KUKA KRL program: MyProgram_303().src

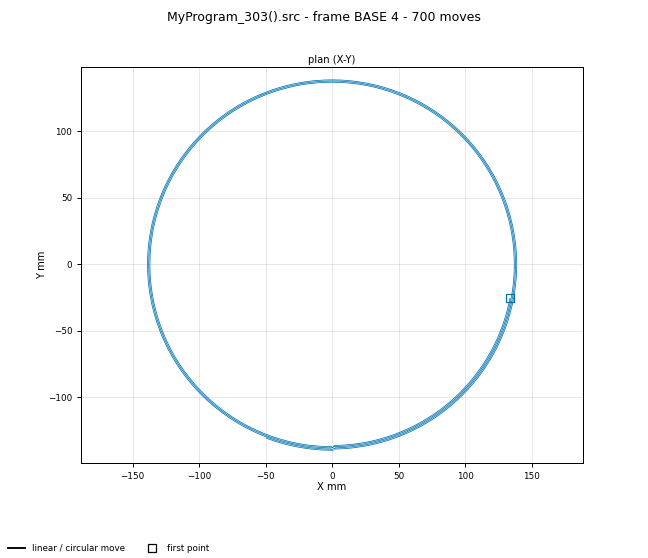
[picture p0: tool path of MyProgram_303().src in frame BASE 4, 700 of 700 moves have a stored position in this frame; points joined in program order, loops and branches not executed]
&ACCESS RVP
&REL 1
&PARAM TEMPLATE = C:\KRC\Roboter\Template\vorgabe
&PARAM EDITMASK = *
DEF MyProgram_303()
; ---- Setting reference (Base) ----
$BASE = BASE_DATA[4]

; --------------------------
; ---- Setting tool (TCP) ----
$TOOL = TOOL_DATA[3]
; --------------------------

$VEL.CP = VEL_APROX_PRINT
Startdeposition()
$VEL.CP = VEL_PRINT
LIN {X 133.6674,Y -25.5337,Z 180,A -8.434,B 5.5878,C 0.2694,E1 5.7512,E2 460.8731} C_DIS
LIN {X 132.8388,Y -29.5533,Z 180,A -10.1187,B 5.5876,C 0.2736,E1 5.7502,E2 462.5539} C_DIS
LIN {X 131.9448,Y -33.3095,Z 180,A -11.8894,B 5.5873,C 0.2804,E1 5.749,E2 464.3442} C_DIS
LIN {X 130.5853,Y -38.2938,Z 180,A -13.8432,B 5.5872,C 0.283,E1 5.7475,E2 466.272} C_DIS
LIN {X 129.5921,Y -41.5309,Z 180,A -15.2343,B 5.587,C 0.2864,E1 5.7464,E2 467.66} C_DIS
LIN {X 127.7254,Y -46.9659,Z 180,A -17.711,B 5.5866,C 0.2938,E1 5.7441,E2 470.1461} C_DIS
LIN {X 125.6978,Y -52.1446,Z 180,A -19.6502,B 5.5866,C 0.294,E1 5.7421,E2 472.0364} C_DIS
LIN {X 124,Y -56.0639,Z 180,A -21.5952,B 5.5862,C 0.3009,E1 5.7399,E2 474.0017} C_DIS
LIN {X 122.3109,Y -59.6596,Z 180,A -23.4453,B 5.5859,C 0.308,E1 5.7376,E2 475.8758} C_DIS
LIN {X 119.5176,Y -65.0767,Z 180,A -25.5702,B 5.5859,C 0.308,E1 5.735,E2 477.947} C_DIS
LIN {X 117.9855,Y -67.8162,Z 180,A -27.1675,B 5.5854,C 0.3154,E1 5.7327,E2 479.5806} C_DIS
LIN {X 115.6089,Y -71.7915,Z 180,A -28.9992,B 5.5853,C 0.3185,E1 5.7301,E2 481.3991} C_DIS
LIN {X 113.3177,Y -75.3564,Z 180,A -30.7531,B 5.585,C 0.3224,E1 5.7274,E2 483.1508} C_DIS
LIN {X 110.9133,Y -78.853,Z 180,A -32.56,B 5.5848,C 0.3269,E1 5.7245,E2 484.9618} C_DIS
LIN {X 108.1869,Y -82.5532,Z 180,A -34.4234,B 5.5846,C 0.3304,E1 5.7214,E2 486.8179} C_DIS
LIN {X 105.3409,Y -86.1552,Z 180,A -36.3118,B 5.5844,C 0.3341,E1 5.7181,E2 488.7023} C_DIS
LIN {X 102.5066,Y -89.5088,Z 180,A -38.1546,B 5.5841,C 0.3382,E1 5.7147,E2 490.546} C_DIS
LIN {X 98.895,Y -93.4837,Z 180,A -40.3296,B 5.5839,C 0.3418,E1 5.7106,E2 492.7121} C_DIS
LIN {X 95.7,Y -96.7524,Z 180,A -42.7451,B 5.5832,C 0.353,E1 5.7057,E2 495.1915} C_DIS
LIN {X 92.0984,Y -100.1859,Z 180,A -44.2158,B 5.5835,C 0.3481,E1 5.7029,E2 496.5848} C_DIS
LIN {X 89.5417,Y -102.4779,Z 180,A -45.5637,B 5.5835,C 0.3495,E1 5.7001,E2 497.9215} C_DIS
LIN {X 86.5764,Y -104.9954,Z 180,A -47.3133,B 5.5831,C 0.3543,E1 5.6963,E2 499.6868} C_DIS
LIN {X 83.034,Y -107.819,Z 180,A -49.2331,B 5.5829,C 0.358,E1 5.6921,E2 501.6099} C_DIS
LIN {X 79.3501,Y -110.5578,Z 180,A -51.1319,B 5.5827,C 0.3609,E1 5.6878,E2 503.5058} C_DIS
LIN {X 75.6563,Y -113.1174,Z 180,A -52.9009,B 5.5826,C 0.3624,E1 5.6838,E2 505.2607} C_DIS
LIN {X 72.317,Y -115.2815,Z 180,A -54.5739,B 5.5824,C 0.3651,E1 5.6798,E2 506.9348} C_DIS
LIN {X 68.7134,Y -117.4647,Z 180,A -56.3441,B 5.5822,C 0.3678,E1 5.6756,E2 508.7059} C_DIS
LIN {X 64.8663,Y -119.6324,Z 180,A -58.2317,B 5.582,C 0.3709,E1 5.6709,E2 510.5987} C_DIS
LIN {X 61.4457,Y -121.4224,Z 180,A -59.7189,B 5.582,C 0.3713,E1 5.6673,E2 512.0694} C_DIS
LIN {X 57.8895,Y -123.1589,Z 180,A -61.3233,B 5.582,C 0.3727,E1 5.6633,E2 513.6671} C_DIS
LIN {X 54.334,Y -124.7671,Z 180,A -63.1891,B 5.5816,C 0.3778,E1 5.6584,E2 515.5626} C_DIS
LIN {X 46.4604,Y -127.9079,Z 180,A -66.358,B 5.5816,C 0.3764,E1 5.6503,E2 518.6828} C_DIS
LIN {X 42.8157,Y -129.1734,Z 180,A -68.124,B 5.5814,C 0.3801,E1 5.6456,E2 520.4682} C_DIS
LIN {X 39.517,Y -130.2207,Z 180,A -69.541,B 5.5814,C 0.3809,E1 5.6418,E2 521.881} C_DIS
LIN {X 36.4352,Y -131.1162,Z 180,A -70.9127,B 5.5813,C 0.3824,E1 5.6381,E2 523.2562} C_DIS
LIN {X 32.8836,Y -132.0529,Z 180,A -72.4265,B 5.5813,C 0.3832,E1 5.634,E2 524.7669} C_DIS
LIN {X 29.4041,Y -132.8715,Z 180,A -74.0382,B 5.581,C 0.3858,E1 5.6296,E2 526.3933} C_DIS
LIN {X 25.5906,Y -133.6566,Z 180,A -75.5921,B 5.581,C 0.3858,E1 5.6254,E2 527.9372} C_DIS
LIN {X 20.5785,Y -134.5197,Z 180,A -77.875,B 5.5808,C 0.3889,E1 5.619,E2 530.2394} C_DIS
LIN {X 17.296,Y -134.9814,Z 180,A -79.1694,B 5.5808,C 0.3883,E1 5.6155,E2 531.5218} C_DIS
LIN {X 8.8845,Y -135.7952,Z 180,A -82.5567,B 5.5809,C 0.3874,E1 5.6061,E2 534.8892} C_DIS
LIN {X 1.7004,Y -136.0752,Z 180,A -85.7728,B 5.5807,C 0.3905,E1 5.5971,E2 538.1311} C_DIS
LIN {X 1.7004,Y -136.0752,Z 180,A -85.7728,B 5.5807,C 0.3905,E1 5.5971,E2 538.1311} C_DIS
Enddeposition()
LIN {X 0.9629,Y -136.9801,Z 180,A -85.7145,B 5.5127,C 0.3881,E1 5.5292,E2 538.0775} C_DIS
Startdeposition()
$VEL.CP = VEL_PRINT
LIN {X 5.9591,Y -136.8588,Z 180,A -82.9076,B 5.5134,C 0.3786,E1 5.5373,E2 535.1764} C_DIS
LIN {X 9.2064,Y -136.6797,Z 180,A -81.1696,B 5.5137,C 0.3733,E1 5.5423,E2 533.388} C_DIS
LIN {X 14.3385,Y -136.2351,Z 180,A -79.6594,B 5.5132,C 0.3808,E1 5.5462,E2 531.9612} C_DIS
LIN {X 22.708,Y -135.0919,Z 180,A -76.1483,B 5.5133,C 0.3792,E1 5.5559,E2 528.4512} C_DIS
LIN {X 26.5585,Y -134.39,Z 180,A -74.4021,B 5.5135,C 0.3767,E1 5.5608,E2 526.6898} C_DIS
LIN {X 30.3798,Y -133.5759,Z 180,A -72.9197,B 5.5135,C 0.3775,E1 5.5648,E2 525.2262} C_DIS
LIN {X 33.4089,Y -132.8509,Z 180,A -71.7147,B 5.5135,C 0.3778,E1 5.568,E2 524.033} C_DIS
LIN {X 36.6138,Y -132.0035,Z 180,A -70.25,B 5.5135,C 0.3756,E1 5.572,E2 522.5573} C_DIS
LIN {X 39.7265,Y -131.1006,Z 180,A -68.8635,B 5.5137,C 0.3739,E1 5.5757,E2 521.1658} C_DIS
LIN {X 43.1088,Y -130.0272,Z 180,A -67.3618,B 5.5137,C 0.3722,E1 5.5797,E2 519.6608} C_DIS
LIN {X 46.2144,Y -128.9561,Z 180,A -64.7574,B 5.515,C 0.3537,E1 5.587,E2 516.8931} C_DIS
LIN {X 54.4369,Y -125.706,Z 180,A -61.9666,B 5.5145,C 0.3619,E1 5.5938,E2 514.2199} C_DIS
LIN {X 58.316,Y -123.9567,Z 180,A -60.5223,B 5.5143,C 0.3642,E1 5.5974,E2 512.8183} C_DIS
LIN {X 61.5186,Y -122.3982,Z 180,A -59.0643,B 5.5144,C 0.3626,E1 5.601,E2 511.3634} C_DIS
LIN {X 65.241,Y -120.4562,Z 180,A -57.3435,B 5.5146,C 0.3606,E1 5.6053,E2 509.6458} C_DIS
LIN {X 68.9644,Y -118.3637,Z 180,A -55.5918,B 5.5147,C 0.3584,E1 5.6095,E2 507.8972} C_DIS
LIN {X 72.6617,Y -116.1305,Z 180,A -53.8371,B 5.5148,C 0.3563,E1 5.6136,E2 506.1478} C_DIS
LIN {X 76.146,Y -113.8758,Z 180,A -52.1006,B 5.515,C 0.3534,E1 5.6177,E2 504.4098} C_DIS
LIN {X 79.7915,Y -111.3519,Z 180,A -50.2937,B 5.5152,C 0.3508,E1 5.6218,E2 502.6076} C_DIS
LIN {X 83.4506,Y -108.637,Z 180,A -48.4066,B 5.5154,C 0.3477,E1 5.626,E2 500.7213} C_DIS
LIN {X 86.9716,Y -105.8394,Z 180,A -46.5374,B 5.5156,C 0.3443,E1 5.6301,E2 498.8521} C_DIS
LIN {X 91.926,Y -101.5655,Z 180,A -43.4145,B 5.5163,C 0.3333,E1 5.6367,E2 495.6763} C_DIS
LIN {X 95.3245,Y -98.3827,Z 180,A -41.896,B 5.5161,C 0.3356,E1 5.6397,E2 494.2123} C_DIS
LIN {X 98.0792,Y -95.6375,Z 180,A -40.532,B 5.5161,C 0.3361,E1 5.6423,E2 492.8809} C_DIS
LIN {X 102.4384,Y -90.9526,Z 180,A -37.732,B 5.5166,C 0.3285,E1 5.6476,E2 490.0626} C_DIS
LIN {X 105.2335,Y -87.7041,Z 180,A -35.9364,B 5.5168,C 0.3244,E1 5.6509,E2 488.2651} C_DIS
LIN {X 108.1029,Y -84.1413,Z 180,A -34.0819,B 5.517,C 0.3209,E1 5.6541,E2 486.4165} C_DIS
LIN {X 110.6826,Y -80.7183,Z 180,A -32.3179,B 5.5172,C 0.3171,E1 5.657,E2 484.6547} C_DIS
LIN {X 113.2996,Y -77.0011,Z 180,A -30.4716,B 5.5174,C 0.3134,E1 5.6599,E2 482.8138} C_DIS
LIN {X 115.7618,Y -73.2472,Z 180,A -28.6372,B 5.5177,C 0.3095,E1 5.6627,E2 480.9833} C_DIS
LIN {X 118.1004,Y -69.4134,Z 180,A -26.8055,B 5.5179,C 0.3055,E1 5.6653,E2 479.1559} C_DIS
LIN {X 120.3903,Y -65.3619,Z 180,A -24.5644,B 5.5184,C 0.2961,E1 5.6684,E2 476.8748} C_DIS
LIN {X 122.2336,Y -61.8418,Z 180,A -23.335,B 5.5183,C 0.2984,E1 5.6699,E2 475.7} C_DIS
LIN {X 124.2076,Y -57.7748,Z 180,A -21.3722,B 5.5186,C 0.2923,E1 5.6722,E2 473.7262} C_DIS
LIN {X 126.0977,Y -53.5294,Z 180,A -19.5105,B 5.5188,C 0.2885,E1 5.6743,E2 471.8735} C_DIS
LIN {X 127.5825,Y -49.8816,Z 180,A -18.0664,B 5.5188,C 0.2872,E1 5.6757,E2 470.4541} C_DIS
LIN {X 128.8042,Y -46.636,Z 180,A -16.4286,B 5.5192,C 0.2804,E1 5.6773,E2 468.7908} C_DIS
LIN {X 130.343,Y -42.1468,Z 180,A -14.6249,B 5.5193,C 0.2777,E1 5.6789,E2 467.0087} C_DIS
LIN {X 131.2957,Y -39.0797,Z 180,A -13.4462,B 5.5193,C 0.2766,E1 5.6799,E2 465.8501} C_DIS
LIN {X 132.2472,Y -35.7252,Z 180,A -12.0475,B 5.5196,C 0.2735,E1 5.6809,E2 464.4578} C_DIS
LIN {X 133.1587,Y -32.1591,Z 180,A -10.4265,B 5.5198,C 0.2679,E1 5.682,E2 462.825} C_DIS
LIN {X 133.9191,Y -28.829,Z 180,A -9.0632,B 5.52,C 0.2649,E1 5.6828,E2 461.4688} C_DIS
LIN {X 135.0379,Y -23.032,Z 180,A -6.3047,B 5.5205,C 0.2535,E1 5.6842,E2 458.6711} C_DIS
LIN {X 135.5799,Y -19.5857,Z 180,A -5.0968,B 5.5205,C 0.2533,E1 5.6847,E2 457.4944} C_DIS
LIN {X 136.2099,Y -14.5726,Z 180,A -2.5529,B 5.5211,C 0.2406,E1 5.6855,E2 454.8933} C_DIS
LIN {X 136.6579,Y -9.505,Z 180,A -1.0891,B 5.5209,C 0.2448,E1 5.6858,E2 453.5132} C_DIS
LIN {X 136.8714,Y -5.6402,Z 180,A 0.5488,B 5.5211,C 0.2399,E1 5.686,E2 451.8716} C_DIS
LIN {X 136.9726,Y -2.0268,Z 180,A 2.7438,B 5.5217,C 0.225,E1 5.6861,E2 449.5877} C_DIS
LIN {X 136.9301,Y 3.962,Z 180,A 4.4252,B 5.5215,C 0.2307,E1 5.6861,E2 448.0102} C_DIS
LIN {X 136.5326,Y 11.157,Z 180,A 7.2664,B 5.5217,C 0.2248,E1 5.6855,E2 445.1889} C_DIS
LIN {X 135.9491,Y 16.8438,Z 180,A 9.7561,B 5.5221,C 0.2165,E1 5.6848,E2 442.685} C_DIS
LIN {X 135.4199,Y 20.6637,Z 180,A 11.3418,B 5.5222,C 0.2123,E1 5.6841,E2 441.1017} C_DIS
LIN {X 134.6933,Y 24.9749,Z 180,A 13.1664,B 5.5224,C 0.2073,E1 5.6832,E2 439.2764} C_DIS
LIN {X 133.926,Y 28.7974,Z 180,A 14.6505,B 5.5225,C 0.205,E1 5.6824,E2 437.8097} C_DIS
LIN {X 133.2251,Y 31.8835,Z 180,A 15.9603,B 5.5226,C 0.2015,E1 5.6816,E2 436.5008} C_DIS
LIN {X 132.3877,Y 35.1986,Z 180,A 17.271,B 5.5227,C 0.1994,E1 5.6807,E2 435.2044} C_DIS
LIN {X 131.4832,Y 38.4392,Z 180,A 18.6758,B 5.5229,C 0.1956,E1 5.6796,E2 433.799} C_DIS
LIN {X 130.378,Y 42.0372,Z 180,A 20.3219,B 5.523,C 0.1902,E1 5.6782,E2 432.1429} C_DIS
LIN {X 129.086,Y 45.8542,Z 180,A 21.9681,B 5.5232,C 0.1863,E1 5.6767,E2 430.5007} C_DIS
LIN {X 127.6955,Y 49.5908,Z 180,A 23.4129,B 5.5232,C 0.1852,E1 5.6753,E2 429.0831} C_DIS
LIN {X 126.4948,Y 52.5784,Z 180,A 24.9531,B 5.5234,C 0.1787,E1 5.6736,E2 427.5177} C_DIS
LIN {X 124.5309,Y 57.0756,Z 180,A 26.8317,B 5.5235,C 0.176,E1 5.6715,E2 425.6601} C_DIS
LIN {X 123.0141,Y 60.2746,Z 180,A 28.2274,B 5.5235,C 0.1735,E1 5.6698,E2 424.2744} C_DIS
LIN {X 121.4029,Y 63.4566,Z 180,A 29.7193,B 5.5237,C 0.1697,E1 5.6679,E2 422.7817} C_DIS
LIN {X 119.27,Y 67.3845,Z 180,A 31.6372,B 5.5239,C 0.1643,E1 5.6653,E2 420.857} C_DIS
LIN {X 117.0777,Y 71.1253,Z 180,A 33.4111,B 5.5239,C 0.1605,E1 5.6628,E2 419.0873} C_DIS
LIN {X 114.7348,Y 74.846,Z 180,A 35.1874,B 5.5241,C 0.157,E1 5.6601,E2 417.3181} C_DIS
LIN {X 112.2574,Y 78.513,Z 180,A 37.0342,B 5.5241,C 0.1527,E1 5.6572,E2 415.4712} C_DIS
LIN {X 109.5754,Y 82.2149,Z 180,A 38.7169,B 5.5242,C 0.1517,E1 5.6544,E2 413.8165} C_DIS
LIN {X 107.2012,Y 85.2866,Z 180,A 40.3892,B 5.5243,C 0.1473,E1 5.6516,E2 412.1376} C_DIS
LIN {X 104.7567,Y 88.2725,Z 180,A 42.0713,B 5.5245,C 0.1428,E1 5.6485,E2 410.4466} C_DIS
LIN {X 101.7751,Y 91.6946,Z 180,A 43.8321,B 5.5245,C 0.1407,E1 5.6453,E2 408.7024} C_DIS
LIN {X 98.7669,Y 94.9271,Z 180,A 45.7626,B 5.5246,C 0.1356,E1 5.6416,E2 406.7611} C_DIS
LIN {X 95.5482,Y 98.1661,Z 180,A 47.3451,B 5.5246,C 0.1364,E1 5.6385,E2 405.2189} C_DIS
LIN {X 92.6799,Y 100.8779,Z 180,A 49.211,B 5.5248,C 0.1302,E1 5.6347,E2 403.3259} C_DIS
LIN {X 89.3728,Y 103.8191,Z 180,A 51.0246,B 5.5248,C 0.1272,E1 5.6309,E2 401.5167} C_DIS
LIN {X 85.8701,Y 106.7346,Z 180,A 52.941,B 5.5249,C 0.1236,E1 5.6267,E2 399.5988} C_DIS
LIN {X 82.2251,Y 109.5677,Z 180,A 54.8506,B 5.5249,C 0.1205,E1 5.6225,E2 397.6917} C_DIS
LIN {X 78.6371,Y 112.1708,Z 180,A 56.653,B 5.525,C 0.1181,E1 5.6184,E2 395.8955} C_DIS
LIN {X 75.107,Y 114.5641,Z 180,A 58.4111,B 5.525,C 0.1156,E1 5.6143,E2 394.1405} C_DIS
LIN {X 71.3198,Y 116.9596,Z 180,A 60.281,B 5.5252,C 0.1128,E1 5.6099,E2 392.2711} C_DIS
LIN {X 67.5354,Y 119.1849,Z 180,A 62.1056,B 5.5252,C 0.1103,E1 5.6055,E2 390.448} C_DIS
LIN {X 63.8288,Y 121.2075,Z 180,A 63.7161,B 5.5252,C 0.11,E1 5.6016,E2 388.8567} C_DIS
LIN {X 61.2437,Y 122.536,Z 180,A 65.023,B 5.5252,C 0.1072,E1 5.5983,E2 387.5387} C_DIS
LIN {X 57.8222,Y 124.1857,Z 180,A 66.5177,B 5.5252,C 0.1064,E1 5.5945,E2 386.0557} C_DIS
LIN {X 54.6205,Y 125.6266,Z 180,A 67.9197,B 5.5252,C 0.1056,E1 5.591,E2 384.662} C_DIS
LIN {X 51.4939,Y 126.9403,Z 180,A 69.2666,B 5.5253,C 0.1049,E1 5.5875,E2 383.3242} C_DIS
LIN {X 48.8881,Y 127.9683,Z 180,A 70.6345,B 5.5253,C 0.1011,E1 5.5839,E2 381.9322} C_DIS
LIN {X 45.08,Y 129.357,Z 180,A 72.0835,B 5.5253,C 0.1027,E1 5.5801,E2 380.5139} C_DIS
LIN {X 42.0821,Y 130.3636,Z 180,A 73.4942,B 5.5253,C 0.1003,E1 5.5764,E2 379.0926} C_DIS
LIN {X 37.472,Y 131.7635,Z 180,A 75.439,B 5.5254,C 0.0995,E1 5.5712,E2 377.1569} C_DIS
LIN {X 33.9468,Y 132.7144,Z 180,A 77.0132,B 5.5254,C 0.0978,E1 5.5669,E2 375.5773} C_DIS
LIN {X 30.7155,Y 133.4992,Z 180,A 78.447,B 5.5254,C 0.0962,E1 5.563,E2 374.1385} C_DIS
LIN {X 27.37,Y 134.2249,Z 180,A 79.87,B 5.5254,C 0.0955,E1 5.5591,E2 372.7169} C_DIS
LIN {X 23.2032,Y 135.0093,Z 180,A 81.6985,B 5.5255,C 0.0938,E1 5.5541,E2 370.8823} C_DIS
LIN {X 19.1357,Y 135.6442,Z 180,A 83.6361,B 5.5255,C 0.0904,E1 5.5487,E2 368.9186} C_DIS
LIN {X 15.5832,Y 136.0995,Z 180,A 85.2933,B 5.5256,C 0.0879,E1 5.544,E2 367.2422} C_DIS
LIN {X 11.3245,Y 136.5185,Z 180,A 86.6921,B 5.5256,C 0.0922,E1 5.5402,E2 365.8924} C_DIS
LIN {X 8.4551,Y 136.7261,Z 180,A 88.5823,B 5.5256,C 0.0836,E1 5.5348,E2 363.9176} C_DIS
LIN {X 2.4594,Y 136.9654,Z 180,A 90.6298,B 5.5256,C 0.0889,E1 5.5292,E2 361.9286} C_DIS
LIN {X -1.0774,Y 136.9835,Z 180,A 91.8821,B 5.5256,C 0.0916,E1 5.5258,E2 360.7051} C_DIS
LIN {X -5.2438,Y 136.8869,Z 180,A 93.5421,B 5.5256,C 0.0927,E1 5.5212,E2 359.056} C_DIS
LIN {X -10.5015,Y 136.5851,Z 180,A 95.9583,B 5.5256,C 0.0905,E1 5.5144,E2 356.6147} C_DIS
LIN {X -16.7957,Y 135.9548,Z 180,A 98.4644,B 5.5256,C 0.0928,E1 5.5074,E2 354.1271} C_DIS
LIN {X -20.631,Y 135.425,Z 180,A 100.0493,B 5.5256,C 0.0938,E1 5.5031,E2 352.5474} C_DIS
LIN {X -24.1026,Y 134.85,Z 180,A 101.5008,B 5.5255,C 0.0947,E1 5.4991,E2 351.0991} C_DIS
LIN {X -27.7276,Y 134.1522,Z 180,A 103.0718,B 5.5255,C 0.0952,E1 5.4948,E2 349.5258} C_DIS
LIN {X -31.8835,Y 133.2251,Z 180,A 104.7738,B 5.5255,C 0.0972,E1 5.4902,E2 347.8345} C_DIS
LIN {X -34.9603,Y 132.4512,Z 180,A 105.9658,B 5.5255,C 0.0996,E1 5.487,E2 346.6599} C_DIS
LIN {X -37.8601,Y 131.6528,Z 180,A 107.5127,B 5.5255,C 0.0973,E1 5.4827,E2 345.0784} C_DIS
LIN {X -41.5721,Y 130.5265,Z 180,A 109.0374,B 5.5255,C 0.0997,E1 5.4787,E2 343.5667} C_DIS
LIN {X -48.3571,Y 128.1682,Z 180,A 112.1227,B 5.5254,C 0.1016,E1 5.4706,E2 340.4736} C_DIS
LIN {X -51.0775,Y 127.1082,Z 180,A 113.5748,B 5.5254,C 0.1004,E1 5.4667,E2 338.9938} C_DIS
LIN {X -55.22,Y 125.3664,Z 180,A 115.3255,B 5.5254,C 0.1038,E1 5.4623,E2 337.2605} C_DIS
LIN {X -58.7178,Y 123.7648,Z 180,A 116.8367,B 5.5253,C 0.1068,E1 5.4585,E2 335.7624} C_DIS
LIN {X -61.8768,Y 122.2159,Z 180,A 118.3402,B 5.5253,C 0.1083,E1 5.4547,E2 334.2561} C_DIS
LIN {X -65.0139,Y 120.5784,Z 180,A 119.9047,B 5.5253,C 0.1093,E1 5.4509,E2 332.6824} C_DIS
LIN {X -68.9535,Y 118.3701,Z 180,A 121.8521,B 5.5252,C 0.1113,E1 5.4461,E2 330.7292} C_DIS
LIN {X -71.6444,Y 116.7604,Z 180,A 123.3661,B 5.5252,C 0.1112,E1 5.4425,E2 329.1912} C_DIS
LIN {X -74.4018,Y 115.0232,Z 180,A 124.5687,B 5.5252,C 0.1149,E1 5.4397,E2 328.0095} C_DIS
LIN {X -77.9872,Y 112.6233,Z 180,A 126.4212,B 5.5251,C 0.1173,E1 5.4354,E2 326.1525} C_DIS
LIN {X -81.7444,Y 109.9262,Z 180,A 128.3434,B 5.525,C 0.1206,E1 5.4311,E2 324.2334} C_DIS
LIN {X -85.3449,Y 107.1549,Z 180,A 130.2501,B 5.525,C 0.1238,E1 5.4269,E2 322.3274} C_DIS
LIN {X -88.6469,Y 104.4397,Z 180,A 132.1044,B 5.5249,C 0.1264,E1 5.4229,E2 320.4664} C_DIS
LIN {X -92.1385,Y 101.3727,Z 180,A 134.0526,B 5.5248,C 0.13,E1 5.4188,E2 318.5193} C_DIS
LIN {X -95.4202,Y 98.29,Z 180,A 135.9744,B 5.5247,C 0.1334,E1 5.4149,E2 316.5944} C_DIS
LIN {X -98.6326,Y 95.0664,Z 180,A 137.9163,B 5.5247,C 0.1368,E1 5.4111,E2 314.6493} C_DIS
LIN {X -101.6556,Y 91.8267,Z 180,A 139.8184,B 5.5245,C 0.1402,E1 5.4075,E2 312.7428} C_DIS
LIN {X -104.4792,Y 88.6004,Z 180,A 141.6551,B 5.5245,C 0.1437,E1 5.4042,E2 310.9022} C_DIS
LIN {X -107.4064,Y 85.0288,Z 180,A 143.6482,B 5.5243,C 0.1474,E1 5.4007,E2 308.9031} C_DIS
LIN {X -110.091,Y 81.5231,Z 180,A 145.5103,B 5.5243,C 0.1514,E1 5.3976,E2 307.0408} C_DIS
LIN {X -112.678,Y 77.9086,Z 180,A 147.4126,B 5.5241,C 0.1553,E1 5.3945,E2 305.1348} C_DIS
LIN {X -114.279,Y 75.54,Z 180,A 148.6489,B 5.5241,C 0.1578,E1 5.3926,E2 303.8945} C_DIS
LIN {X -117.1143,Y 71.0648,Z 180,A 150.8875,B 5.5239,C 0.1629,E1 5.3893,E2 301.655} C_DIS
LIN {X -119.3249,Y 67.2869,Z 180,A 152.7732,B 5.5238,C 0.167,E1 5.3866,E2 299.7641} C_DIS
LIN {X -121.5025,Y 63.267,Z 180,A 155.0178,B 5.5238,C 0.1687,E1 5.3837,E2 297.4796} C_DIS
LIN {X -123.2185,Y 59.8602,Z 180,A 156.3404,B 5.5235,C 0.1753,E1 5.3821,E2 296.1927} C_DIS
LIN {X -124.8727,Y 56.3238,Z 180,A 157.9398,B 5.5234,C 0.1798,E1 5.3802,E2 294.5988} C_DIS
LIN {X -126.2063,Y 53.2692,Z 180,A 159.4289,B 5.5233,C 0.1826,E1 5.3786,E2 293.0991} C_DIS
LIN {X -127.6676,Y 49.6625,Z 180,A 161.0329,B 5.5231,C 0.1872,E1 5.3769,E2 291.4994} C_DIS
LIN {X -130.2229,Y 42.521,Z 180,A 164.4398,B 5.5229,C 0.1936,E1 5.3738,E2 288.0662} C_DIS
LIN {X -132.1707,Y 36.0121,Z 180,A 167.3523,B 5.5227,C 0.2008,E1 5.3715,E2 285.1473} C_DIS
LIN {X -133.1847,Y 32.0508,Z 180,A 168.8875,B 5.5224,C 0.2071,E1 5.3705,E2 283.6354} C_DIS
LIN {X -133.8797,Y 29.0117,Z 180,A 170.3023,B 5.5224,C 0.2097,E1 5.3696,E2 282.2078} C_DIS
LIN {X -134.5787,Y 25.5743,Z 180,A 171.826,B 5.5222,C 0.2133,E1 5.3688,E2 280.6782} C_DIS
LIN {X -135.3067,Y 21.3955,Z 180,A 173.6561,B 5.522,C 0.2178,E1 5.368,E2 278.8427} C_DIS
LIN {X -135.7841,Y 18.1179,Z 180,A 175.094,B 5.5219,C 0.2212,E1 5.3674,E2 277.3993} C_DIS
LIN {X -136.2011,Y 14.6539,Z 180,A 176.5536,B 5.5217,C 0.2254,E1 5.3669,E2 275.9408} C_DIS
LIN {X -136.5505,Y 10.9457,Z 180,A 178.2214,B 5.5216,C 0.2288,E1 5.3665,E2 274.2605} C_DIS
LIN {X -136.8207,Y 6.7542,Z 180,A 179.9883,B 5.5214,C 0.2337,E1 5.3663,E2 272.4936} C_DIS
LIN {X -136.9645,Y 2.5098,Z 180,A -178.198,B 5.5212,C 0.2385,E1 5.3661,E2 270.6767} C_DIS
LIN {X -136.9795,Y -1.6063,Z 180,A -176.3484,B 5.521,C 0.2422,E1 5.3661,E2 268.8123} C_DIS
LIN {X -136.8732,Y -5.5952,Z 180,A -174.6513,B 5.5208,C 0.2467,E1 5.3663,E2 267.1127} C_DIS
LIN {X -136.6367,Y -9.7954,Z 180,A -172.9278,B 5.5206,C 0.252,E1 5.3666,E2 265.3951} C_DIS
LIN {X -136.3486,Y -13.2123,Z 180,A -171.4508,B 5.5204,C 0.2557,E1 5.367,E2 263.9137} C_DIS
LIN {X -135.9321,Y -16.9858,Z 180,A -169.7822,B 5.5202,C 0.2595,E1 5.3675,E2 262.2361} C_DIS
LIN {X -135.4106,Y -20.7242,Z 180,A -168.1633,B 5.52,C 0.2635,E1 5.3682,E2 260.6132} C_DIS
LIN {X -134.8324,Y -24.201,Z 180,A -166.6195,B 5.5199,C 0.267,E1 5.3689,E2 259.0616} C_DIS
LIN {X -133.9847,Y -28.5252,Z 180,A -164.7599,B 5.5196,C 0.272,E1 5.37,E2 257.2011} C_DIS
LIN {X -133.2114,Y -31.9403,Z 180,A -163.083,B 5.5196,C 0.2741,E1 5.3711,E2 255.4982} C_DIS
LIN {X -131.3234,Y -38.985,Z 180,A -160.0565,B 5.5191,C 0.2826,E1 5.3733,E2 252.4767} C_DIS
LIN {X -130.053,Y -43.0312,Z 180,A -158.5073,B 5.5187,C 0.2895,E1 5.3746,E2 250.9571} C_DIS
LIN {X -128.3114,Y -47.9748,Z 180,A -156.0573,B 5.5186,C 0.2929,E1 5.377,E2 248.4756} C_DIS
LIN {X -127.1245,Y -51.0369,Z 180,A -154.6333,B 5.5184,C 0.296,E1 5.3784,E2 247.0459} C_DIS
LIN {X -125.7124,Y -54.4222,Z 180,A -153.1744,B 5.5181,C 0.3007,E1 5.38,E2 245.5974} C_DIS
LIN {X -124.3954,Y -57.3686,Z 180,A -151.6856,B 5.5181,C 0.3029,E1 5.3818,E2 244.0916} C_DIS
LIN {X -122.5724,Y -61.17,Z 180,A -149.85,B 5.5178,C 0.3066,E1 5.384,E2 242.2477} C_DIS
LIN {X -120.6186,Y -64.939,Z 180,A -148.0859,B 5.5176,C 0.3111,E1 5.3863,E2 240.4858} C_DIS
LIN {X -118.3791,Y -68.9379,Z 180,A -146.0638,B 5.5174,C 0.3148,E1 5.3891,E2 238.4512} C_DIS
LIN {X -116.1088,Y -72.6967,Z 180,A -144.1651,B 5.5171,C 0.3186,E1 5.3919,E2 236.5453} C_DIS
LIN {X -113.6973,Y -76.4135,Z 180,A -142.2344,B 5.5169,C 0.3221,E1 5.3949,E2 234.6054} C_DIS
LIN {X -111.1285,Y -80.1031,Z 180,A -140.3205,B 5.5167,C 0.326,E1 5.398,E2 232.6878} C_DIS
LIN {X -108.3692,Y -83.7977,Z 180,A -138.3801,B 5.5165,C 0.3302,E1 5.4013,E2 230.7466} C_DIS
LIN {X -105.4348,Y -87.461,Z 180,A -136.3998,B 5.5162,C 0.3342,E1 5.4048,E2 228.7647} C_DIS
LIN {X -102.7591,Y -90.5898,Z 180,A -134.1066,B 5.5163,C 0.332,E1 5.4092,E2 226.3979} C_DIS
LIN {X -99.379,Y -94.2859,Z 180,A -132.4987,B 5.5158,C 0.3412,E1 5.4121,E2 224.8538} C_DIS
LIN {X -96.1662,Y -97.5607,Z 180,A -130.5157,B 5.5156,C 0.3443,E1 5.416,E2 222.8629} C_DIS
LIN {X -93.0223,Y -100.5632,Z 180,A -128.6509,B 5.5154,C 0.3472,E1 5.4198,E2 220.9924} C_DIS
LIN {X -90.2215,Y -103.0826,Z 180,A -126.9158,B 5.5154,C 0.3484,E1 5.4235,E2 219.237} C_DIS
LIN {X -86.1573,Y -106.5029,Z 180,A -124.839,B 5.515,C 0.3537,E1 5.428,E2 217.1793} C_DIS
LIN {X -82.6996,Y -109.2096,Z 180,A -122.9697,B 5.5148,C 0.3564,E1 5.4321,E2 215.3059} C_DIS
LIN {X -79.1565,Y -111.8044,Z 180,A -121.121,B 5.5147,C 0.3592,E1 5.4363,E2 213.4558} C_DIS
LIN {X -75.775,Y -114.1235,Z 180,A -119.3511,B 5.5145,C 0.3612,E1 5.4404,E2 211.6788} C_DIS
LIN {X -72.1149,Y -116.4708,Z 180,A -117.5251,B 5.5144,C 0.3637,E1 5.4447,E2 209.852} C_DIS
LIN {X -68.2672,Y -118.7674,Z 180,A -115.5976,B 5.5142,C 0.3656,E1 5.4494,E2 207.9175} C_DIS
LIN {X -64.39,Y -120.9129,Z 180,A -113.7925,B 5.514,C 0.3685,E1 5.4538,E2 206.1186} C_DIS
LIN {X -61.2254,Y -122.5451,Z 180,A -112.2197,B 5.514,C 0.3693,E1 5.4578,E2 204.5348} C_DIS
LIN {X -57.8098,Y -124.1914,Z 180,A -110.7347,B 5.5138,C 0.3722,E1 5.4615,E2 203.0628} C_DIS
LIN {X -54.9048,Y -125.5037,Z 180,A -109.3801,B 5.5138,C 0.3733,E1 5.4649,E2 201.7053} C_DIS
LIN {X -52.0165,Y -126.7289,Z 180,A -107.9405,B 5.5138,C 0.3732,E1 5.4687,E2 200.249} C_DIS
LIN {X -48.2267,Y -128.217,Z 180,A -106.4581,B 5.5135,C 0.3772,E1 5.4725,E2 198.7949} C_DIS
LIN {X -45.7391,Y -129.1275,Z 180,A -105.0653,B 5.5136,C 0.3749,E1 5.4763,E2 197.3648} C_DIS
LIN {X -40.6777,Y -130.8094,Z 180,A -103.0524,B 5.5133,C 0.3791,E1 5.4815,E2 195.3799} C_DIS
LIN {X -37.0885,Y -131.8708,Z 180,A -101.3685,B 5.5133,C 0.3788,E1 5.4861,E2 193.6802} C_DIS
LIN {X -33.9468,Y -132.7144,Z 180,A -99.9951,B 5.5133,C 0.3795,E1 5.4898,E2 192.3047} C_DIS
LIN {X -30.5974,Y -133.5262,Z 180,A -98.5685,B 5.5133,C 0.3804,E1 5.4937,E2 190.8797} C_DIS
LIN {X -26.8584,Y -134.329,Z 180,A -96.8584,B 5.5133,C 0.3798,E1 5.4984,E2 189.1547} C_DIS
LIN {X -23.1372,Y -135.0203,Z 180,A -94.9328,B 5.5135,C 0.3762,E1 5.5038,E2 187.1838} C_DIS
LIN {X -19.0269,Y -135.6598,Z 180,A -93.5267,B 5.5132,C 0.3808,E1 5.5076,E2 185.8207} C_DIS
LIN {X -14.7911,Y -136.1864,Z 180,A -91.8602,B 5.5131,C 0.3826,E1 5.5122,E2 184.1691} C_DIS
LIN {X -8.7636,Y -136.7071,Z 180,A -89.1656,B 5.5132,C 0.3808,E1 5.5198,E2 181.4521} C_DIS
LIN {X -3.9799,Y -136.9296,Z 180,A -87.3425,B 5.5131,C 0.3831,E1 5.5248,E2 179.6516} C_DIS
LIN {X -0.5118,Y -136.9866,Z 180,A -85.7833,B 5.5131,C 0.3815,E1 5.5292,E2 178.0775} C_DIS
LIN {X -0.5118,Y -136.9866,Z 180,A -85.7833,B 5.5131,C 0.3815,E1 5.5292,E2 178.0775} C_DIS
Enddeposition()
LIN {X 0.9731,Y -137.885,Z 180,A -85.2998,B 5.4467,C 0.3854,E1 5.4643,E2 177.6628} C_DIS
Startdeposition()
$VEL.CP = VEL_PRINT
LIN {X -2.4494,Y -137.8683,Z 180,A -87.2819,B 5.4462,C 0.3925,E1 5.4585,E2 179.7189} C_DIS
LIN {X -6.1473,Y -137.755,Z 180,A -88.7568,B 5.4462,C 0.3918,E1 5.4544,E2 181.1864} C_DIS
LIN {X -9.2578,Y -137.581,Z 180,A -90.0542,B 5.4462,C 0.3918,E1 5.4508,E2 182.4847} C_DIS
LIN {X -13.3319,Y -137.2439,Z 180,A -91.7985,B 5.4462,C 0.3921,E1 5.4459,E2 184.2356} C_DIS
LIN {X -17.1247,Y -136.8246,Z 180,A -93.3499,B 5.4462,C 0.3914,E1 5.4416,E2 185.7833} C_DIS
LIN {X -20.3016,Y -136.3894,Z 180,A -94.688,B 5.4462,C 0.3911,E1 5.4379,E2 187.1225} C_DIS
LIN {X -23.4919,Y -135.8763,Z 180,A -96.0371,B 5.4462,C 0.3907,E1 5.4342,E2 188.473} C_DIS
LIN {X -26.1819,Y -135.3816,Z 180,A -97.2269,B 5.4462,C 0.3909,E1 5.4309,E2 189.67} C_DIS
LIN {X -29.9023,Y -134.6109,Z 180,A -98.768,B 5.4464,C 0.3897,E1 5.4267,E2 191.2068} C_DIS
LIN {X -33.1168,Y -133.8563,Z 180,A -100.1492,B 5.4464,C 0.389,E1 5.4229,E2 192.5894} C_DIS
LIN {X -36.093,Y -133.0833,Z 180,A -101.4205,B 5.4464,C 0.3882,E1 5.4195,E2 193.8603} C_DIS
LIN {X -39.55,Y -132.0986,Z 180,A -102.9413,B 5.4465,C 0.3875,E1 5.4154,E2 195.385} C_DIS
LIN {X -42.7627,Y -131.0938,Z 180,A -104.3516,B 5.4465,C 0.3866,E1 5.4117,E2 196.7971} C_DIS
LIN {X -45.9685,Y -130.0044,Z 180,A -105.7711,B 5.4466,C 0.3856,E1 5.4079,E2 198.2185} C_DIS
LIN {X -48.7145,Y -128.9982,Z 180,A -106.9979,B 5.4467,C 0.3846,E1 5.4047,E2 199.4469} C_DIS
LIN {X -52.3467,Y -127.5698,Z 180,A -108.6359,B 5.4468,C 0.3833,E1 5.4004,E2 201.0873} C_DIS
LIN {X -55.5127,Y -126.2243,Z 180,A -110.0807,B 5.4468,C 0.382,E1 5.3967,E2 202.5343} C_DIS
LIN {X -58.1961,Y -125.0073,Z 180,A -111.3622,B 5.4469,C 0.3813,E1 5.3935,E2 203.8233} C_DIS
LIN {X -61.7815,Y -123.2773,Z 180,A -112.9924,B 5.4471,C 0.3791,E1 5.3894,E2 205.4506} C_DIS
LIN {X -64.4484,Y -121.9017,Z 180,A -114.2005,B 5.4472,C 0.3772,E1 5.3864,E2 206.6537} C_DIS
LIN {X -67.9438,Y -119.9912,Z 180,A -116.0129,B 5.4472,C 0.3768,E1 5.3819,E2 208.4865} C_DIS
LIN {X -71.7292,Y -117.7674,Z 180,A -117.8623,B 5.4474,C 0.3746,E1 5.3775,E2 210.3392} C_DIS
LIN {X -75.4559,Y -115.4151,Z 180,A -119.7284,B 5.4476,C 0.3723,E1 5.3731,E2 212.2098} C_DIS
LIN {X -79.1176,Y -112.9365,Z 180,A -121.6174,B 5.4477,C 0.37,E1 5.3687,E2 214.1053} C_DIS
LIN {X -82.7078,Y -110.3343,Z 180,A -123.4818,B 5.4479,C 0.3673,E1 5.3645,E2 215.9725} C_DIS
LIN {X -86.2205,Y -107.6117,Z 180,A -125.3659,B 5.4481,C 0.3646,E1 5.3604,E2 217.8611} C_DIS
LIN {X -89.6495,Y -104.7721,Z 180,A -127.2146,B 5.4483,C 0.3614,E1 5.3564,E2 219.7094} C_DIS
LIN {X -92.9893,Y -101.8196,Z 180,A -129.1321,B 5.4485,C 0.3586,E1 5.3524,E2 221.6349} C_DIS
LIN {X -96.2342,Y -98.7583,Z 180,A -131.0195,B 5.4487,C 0.3555,E1 5.3486,E2 223.5263} C_DIS
LIN {X -99.3464,Y -95.6268,Z 180,A -132.8606,B 5.4489,C 0.3519,E1 5.345,E2 225.3678} C_DIS
LIN {X -102.4189,Y -92.3288,Z 180,A -134.7967,B 5.4491,C 0.3488,E1 5.3414,E2 227.3116} C_DIS
LIN {X -105.3492,Y -88.9707,Z 180,A -136.6529,B 5.4494,C 0.3449,E1 5.338,E2 229.1678} C_DIS
LIN {X -108.1657,Y -85.5244,Z 180,A -138.5723,B 5.4496,C 0.3416,E1 5.3346,E2 231.0956} C_DIS
LIN {X -110.8645,Y -81.9958,Z 180,A -140.4238,B 5.4498,C 0.3376,E1 5.3315,E2 232.9472} C_DIS
LIN {X -113.4422,Y -78.3907,Z 180,A -142.3043,B 5.4501,C 0.3338,E1 5.3285,E2 234.832} C_DIS
LIN {X -115.8957,Y -74.7156,Z 180,A -144.1631,B 5.4503,C 0.3297,E1 5.3256,E2 236.693} C_DIS
LIN {X -118.2225,Y -70.9766,Z 180,A -146.0824,B 5.4505,C 0.3262,E1 5.3228,E2 238.623} C_DIS
LIN {X -120.4203,Y -67.1803,Z 180,A -147.9459,B 5.4508,C 0.3221,E1 5.3202,E2 240.4908} C_DIS
LIN {X -122.4874,Y -63.3331,Z 180,A -149.6874,B 5.4511,C 0.3169,E1 5.318,E2 242.2221} C_DIS
LIN {X -123.9502,Y -60.4173,Z 180,A -151.0834,B 5.4512,C 0.3139,E1 5.3162,E2 243.6226} C_DIS
LIN {X -125.5195,Y -57.0884,Z 180,A -152.6394,B 5.4514,C 0.3103,E1 5.3144,E2 245.1813} C_DIS
LIN {X -126.9012,Y -53.9472,Z 180,A -154.0993,B 5.4516,C 0.3069,E1 5.3128,E2 246.6448} C_DIS
LIN {X -128.2105,Y -50.7574,Z 180,A -155.566,B 5.4518,C 0.3035,E1 5.3113,E2 248.1151} C_DIS
LIN {X -129.4277,Y -47.5678,Z 180,A -157.019,B 5.452,C 0.3,E1 5.3098,E2 249.5716} C_DIS
LIN {X -130.5597,Y -44.3666,Z 180,A -158.4642,B 5.4522,C 0.2966,E1 5.3085,E2 251.0204} C_DIS
LIN {X -131.5271,Y -41.4064,Z 180,A -159.803,B 5.4524,C 0.2935,E1 5.3074,E2 252.364} C_DIS
LIN {X -132.5693,Y -37.9421,Z 180,A -161.3302,B 5.4526,C 0.2896,E1 5.3061,E2 253.8934} C_DIS
LIN {X -133.4481,Y -34.7252,Z 180,A -162.7503,B 5.4528,C 0.2862,E1 5.3051,E2 255.317} C_DIS
LIN {X -134.1513,Y -31.893,Z 180,A -164.015,B 5.4529,C 0.2833,E1 5.3043,E2 256.5875} C_DIS
LIN {X -134.9575,Y -28.2968,Z 180,A -165.5628,B 5.4531,C 0.2792,E1 5.3034,E2 258.1364} C_DIS
LIN {X -135.5871,Y -25.1068,Z 180,A -166.9475,B 5.4533,C 0.2757,E1 5.3026,E2 259.5244} C_DIS
LIN {X -136.1103,Y -22.0893,Z 180,A -168.2236,B 5.4535,C 0.2722,E1 5.302,E2 260.8001} C_DIS
LIN {X -136.5261,Y -19.3451,Z 180,A -169.4342,B 5.4536,C 0.2695,E1 5.3016,E2 262.0171} C_DIS
LIN {X -136.9382,Y -16.1729,Z 180,A -170.797,B 5.4538,C 0.266,E1 5.3011,E2 263.3832} C_DIS
LIN {X -137.3097,Y -12.6471,Z 180,A -172.271,B 5.454,C 0.2619,E1 5.3007,E2 264.8563} C_DIS
LIN {X -137.5473,Y -9.7197,Z 180,A -173.548,B 5.4541,C 0.2589,E1 5.3004,E2 266.1396} C_DIS
LIN {X -137.755,Y -6.1473,Z 180,A -175.0844,B 5.4543,C 0.2551,E1 5.3002,E2 267.6811} C_DIS
LIN {X -137.8837,Y -1.527,Z 180,A -176.9911,B 5.4545,C 0.2495,E1 5.3,E2 269.5847} C_DIS
LIN {X -137.8837,Y 1.527,Z 180,A -178.3583,B 5.4547,C 0.2468,E1 5.3,E2 270.9633} C_DIS
LIN {X -137.7771,Y 5.5821,Z 180,A 179.848,B 5.4548,C 0.2429,E1 5.3002,E2 272.7691} C_DIS
LIN {X -137.581,Y 9.2578,Z 180,A 178.332,B 5.455,C 0.2385,E1 5.3005,E2 274.2823} C_DIS
LIN {X -137.2435,Y 13.3367,Z 180,A 176.5649,B 5.4552,C 0.2342,E1 5.3009,E2 276.0563} C_DIS
LIN {X -136.9028,Y 16.4697,Z 180,A 175.1989,B 5.4554,C 0.231,E1 5.3013,E2 277.4283} C_DIS
LIN {X -136.4069,Y 20.1794,Z 180,A 173.6481,B 5.4555,C 0.2266,E1 5.3019,E2 278.9774} C_DIS
LIN {X -135.8763,Y 23.4919,Z 180,A 172.1992,B 5.4557,C 0.2231,E1 5.3026,E2 280.4319} C_DIS
LIN {X -135.2838,Y 26.693,Z 180,A 170.8077,B 5.4558,C 0.2197,E1 5.3033,E2 281.8272} C_DIS
LIN {X -134.7056,Y 29.4636,Z 180,A 169.5612,B 5.4559,C 0.217,E1 5.3041,E2 283.0815} C_DIS
LIN {X -133.8563,Y 33.1168,Z 180,A 167.9957,B 5.4561,C 0.2128,E1 5.3051,E2 284.6466} C_DIS
LIN {X -133.0192,Y 36.3337,Z 180,A 166.5758,B 5.4562,C 0.2093,E1 5.3061,E2 286.0702} C_DIS
LIN {X -132.1757,Y 39.2868,Z 180,A 165.2651,B 5.4564,C 0.2061,E1 5.3071,E2 287.384} C_DIS
LIN {X -131.0938,Y 42.7627,Z 180,A 163.7099,B 5.4564,C 0.2024,E1 5.3085,E2 288.9433} C_DIS
LIN {X -130.0876,Y 45.7285,Z 180,A 162.3602,B 5.4566,C 0.1993,E1 5.3097,E2 290.2977} C_DIS
LIN {X -128.8298,Y 49.1642,Z 180,A 160.8116,B 5.4567,C 0.1955,E1 5.3112,E2 291.8486} C_DIS
LIN {X -127.5698,Y 52.3467,Z 180,A 159.3518,B 5.4569,C 0.1921,E1 5.3127,E2 293.3118} C_DIS
LIN {X -126.4513,Y 54.9876,Z 180,A 158.121,B 5.4569,C 0.1893,E1 5.3141,E2 294.5464} C_DIS
LIN {X -124.7934,Y 58.6587,Z 180,A 156.4115,B 5.4571,C 0.1853,E1 5.3161,E2 296.2589} C_DIS
LIN {X -123.3135,Y 61.708,Z 180,A 154.9656,B 5.4572,C 0.182,E1 5.3179,E2 297.7082} C_DIS
LIN {X -121.6763,Y 64.8776,Z 180,A 153.5189,B 5.4573,C 0.1779,E1 5.3198,E2 299.1492} C_DIS
LIN {X -120.0252,Y 67.8832,Z 180,A 151.8966,B 5.4574,C 0.1762,E1 5.322,E2 300.7947} C_DIS
LIN {X -117.7674,Y 71.7292,Z 180,A 150.0061,B 5.4575,C 0.172,E1 5.3247,E2 302.6882} C_DIS
LIN {X -115.4151,Y 75.4559,Z 180,A 148.1357,B 5.4577,C 0.168,E1 5.3275,E2 304.5618} C_DIS
LIN {X -112.9365,Y 79.1176,Z 180,A 146.2187,B 5.4577,C 0.1644,E1 5.3306,E2 306.487} C_DIS
LIN {X -110.3343,Y 82.7078,Z 180,A 144.3539,B 5.4579,C 0.1604,E1 5.3337,E2 308.3529} C_DIS
LIN {X -107.6117,Y 86.2205,Z 180,A 142.4477,B 5.4579,C 0.1568,E1 5.337,E2 310.2648} C_DIS
LIN {X -104.7721,Y 89.6495,Z 180,A 140.5916,B 5.4581,C 0.1529,E1 5.3403,E2 312.1201} C_DIS
LIN {X -101.8196,Y 92.9893,Z 180,A 138.6845,B 5.4581,C 0.1495,E1 5.3439,E2 314.0324} C_DIS
LIN {X -98.7583,Y 96.2342,Z 180,A 136.7986,B 5.4583,C 0.146,E1 5.3475,E2 315.9207} C_DIS
LIN {X -95.5931,Y 99.3791,Z 180,A 134.9224,B 5.4583,C 0.1425,E1 5.3513,E2 317.7981} C_DIS
LIN {X -92.3288,Y 102.4189,Z 180,A 133.0204,B 5.4585,C 0.1394,E1 5.3552,E2 319.7044} C_DIS
LIN {X -88.9707,Y 105.3492,Z 180,A 131.1515,B 5.4585,C 0.1362,E1 5.3592,E2 321.5739} C_DIS
LIN {X -85.5244,Y 108.1657,Z 180,A 129.239,B 5.4586,C 0.1336,E1 5.3633,E2 323.4926} C_DIS
LIN {X -81.9958,Y 110.8645,Z 180,A 127.3968,B 5.4586,C 0.1304,E1 5.3674,E2 325.3329} C_DIS
LIN {X -78.3907,Y 113.4422,Z 180,A 125.5281,B 5.4587,C 0.1277,E1 5.3717,E2 327.2035} C_DIS
LIN {X -74.7156,Y 115.8957,Z 180,A 123.6698,B 5.4588,C 0.1251,E1 5.3761,E2 329.063} C_DIS
LIN {X -70.9766,Y 118.2225,Z 180,A 121.7804,B 5.4588,C 0.123,E1 5.3806,E2 330.9583} C_DIS
LIN {X -67.1803,Y 120.4203,Z 180,A 119.9356,B 5.4589,C 0.1207,E1 5.3851,E2 332.8045} C_DIS
LIN {X -63.3331,Y 122.4874,Z 180,A 118.2138,B 5.4589,C 0.1174,E1 5.3893,E2 334.5136} C_DIS
LIN {X -60.2232,Y 124.046,Z 180,A 116.7527,B 5.459,C 0.1158,E1 5.3929,E2 335.9755} C_DIS
LIN {X -57.3427,Y 125.4019,Z 180,A 115.402,B 5.459,C 0.1145,E1 5.3964,E2 337.3285} C_DIS
LIN {X -53.932,Y 126.9077,Z 180,A 113.8526,B 5.459,C 0.1128,E1 5.4003,E2 338.8769} C_DIS
LIN {X -50.7574,Y 128.2105,Z 180,A 112.4148,B 5.4591,C 0.1115,E1 5.4041,E2 340.3153} C_DIS
LIN {X -47.5678,Y 129.4277,Z 180,A 110.9847,B 5.4591,C 0.1102,E1 5.4078,E2 341.7458} C_DIS
LIN {X -44.3666,Y 130.5597,Z 180,A 109.5636,B 5.4591,C 0.1091,E1 5.4116,E2 343.1672} C_DIS
LIN {X -41.3094,Y 131.5581,Z 180,A 108.2135,B 5.4591,C 0.1081,E1 5.4152,E2 344.5181} C_DIS
LIN {X -37.9421,Y 132.5693,Z 180,A 106.7491,B 5.4591,C 0.107,E1 5.4191,E2 345.9821} C_DIS
LIN {X -35.0506,Y 133.3613,Z 180,A 105.4788,B 5.4592,C 0.1064,E1 5.4225,E2 347.2545} C_DIS
LIN {X -31.7997,Y 134.1738,Z 180,A 104.0814,B 5.4592,C 0.1056,E1 5.4263,E2 348.6517} C_DIS
LIN {X -28.2968,Y 134.9575,Z 180,A 102.6011,B 5.4592,C 0.1046,E1 5.4303,E2 350.1299} C_DIS
LIN {X -25.0913,Y 135.5901,Z 180,A 101.2392,B 5.4592,C 0.104,E1 5.4341,E2 351.4915} C_DIS
LIN {X -21.8952,Y 136.1427,Z 180,A 99.8883,B 5.4592,C 0.1034,E1 5.4378,E2 352.8421} C_DIS
LIN {X -17.7571,Y 136.7418,Z 180,A 98.106,B 5.4592,C 0.1034,E1 5.4427,E2 354.6288} C_DIS
LIN {X -13.9639,Y 137.1833,Z 180,A 96.5601,B 5.4592,C 0.1024,E1 5.447,E2 356.1689} C_DIS
LIN {X -10.8214,Y 137.4668,Z 180,A 95.2489,B 5.4592,C 0.1022,E1 5.4507,E2 357.4795} C_DIS
LIN {X -7.6997,Y 137.677,Z 180,A 93.9495,B 5.4592,C 0.102,E1 5.4543,E2 358.7782} C_DIS
LIN {X -3.6745,Y 137.8411,Z 180,A 92.2137,B 5.4592,C 0.1026,E1 5.4592,E2 360.5207} C_DIS
LIN {X -0.6086,Y 137.8887,Z 180,A 90.9416,B 5.4592,C 0.1026,E1 5.4627,E2 361.792} C_DIS
LIN {X 2.4494,Y 137.8683,Z 180,A 89.6687,B 5.4592,C 0.1026,E1 5.4663,E2 363.0647} C_DIS
LIN {X 6.1473,Y 137.755,Z 180,A 88.1961,B 5.4592,C 0.1022,E1 5.4703,E2 364.5288} C_DIS
LIN {X 10.044,Y 137.5236,Z 180,A 86.5472,B 5.4592,C 0.1028,E1 5.475,E2 366.1802} C_DIS
LIN {X 13.3367,Y 137.2435,Z 180,A 85.1798,B 5.4592,C 0.1032,E1 5.4788,E2 367.5464} C_DIS
LIN {X 17.1247,Y 136.8246,Z 180,A 83.6209,B 5.4592,C 0.1035,E1 5.4831,E2 369.1018} C_DIS
LIN {X 20.3016,Y 136.3894,Z 180,A 82.2918,B 5.4592,C 0.104,E1 5.4867,E2 370.4301} C_DIS
LIN {X 23.1578,Y 135.932,Z 180,A 81.0716,B 5.4592,C 0.1048,E1 5.4901,E2 371.6521} C_DIS
LIN {X 26.693,Y 135.2838,Z 180,A 79.6055,B 5.4592,C 0.1054,E1 5.4941,E2 373.1144} C_DIS
LIN {X 29.9023,Y 134.6109,Z 180,A 78.249,B 5.4592,C 0.1062,E1 5.4978,E2 374.4699} C_DIS
LIN {X 32.8818,Y 133.913,Z 180,A 76.9997,B 5.4592,C 0.1068,E1 5.5012,E2 375.7161} C_DIS
LIN {X 36.3337,Y 133.0192,Z 180,A 75.5106,B 5.4592,C 0.108,E1 5.5052,E2 377.2059} C_DIS
LIN {X 39.55,Y 132.0986,Z 180,A 74.1292,B 5.4592,C 0.109,E1 5.5089,E2 378.5858} C_DIS
LIN {X 42.7627,Y 131.0938,Z 180,A 72.7405,B 5.4592,C 0.1102,E1 5.5126,E2 379.9731} C_DIS
LIN {X 45.6027,Y 130.1312,Z 180,A 71.5029,B 5.4592,C 0.1113,E1 5.5159,E2 381.2094} C_DIS
LIN {X 49.1642,Y 128.8298,Z 180,A 69.9413,B 5.4591,C 0.1127,E1 5.52,E2 382.7691} C_DIS
LIN {X 52.3467,Y 127.5698,Z 180,A 68.5321,B 5.4591,C 0.1141,E1 5.5236,E2 384.1765} C_DIS
LIN {X 55.0796,Y 126.4116,Z 180,A 67.2731,B 5.4591,C 0.1158,E1 5.5269,E2 385.4385} C_DIS
LIN {X 58.6587,Y 124.7934,Z 180,A 65.6952,B 5.459,C 0.1171,E1 5.5308,E2 387.0096} C_DIS
LIN {X 61.5857,Y 123.3739,Z 180,A 64.3491,B 5.459,C 0.1188,E1 5.5342,E2 388.3548} C_DIS
LIN {X 64.6198,Y 121.8117,Z 180,A 63.0282,B 5.459,C 0.1194,E1 5.5375,E2 389.6637} C_DIS
LIN {X 67.9438,Y 119.9912,Z 180,A 61.3213,B 5.4588,C 0.1234,E1 5.5417,E2 391.3869} C_DIS
LIN {X 71.7292,Y 117.7674,Z 180,A 59.5205,B 5.4588,C 0.1258,E1 5.546,E2 393.1849} C_DIS
LIN {X 75.4559,Y 115.4151,Z 180,A 57.6828,B 5.4588,C 0.1287,E1 5.5503,E2 395.0235} C_DIS
LIN {X 79.1176,Y 112.9365,Z 180,A 55.9137,B 5.4587,C 0.1308,E1 5.5543,E2 396.7842} C_DIS
LIN {X 82.7078,Y 110.3343,Z 180,A 54.0573,B 5.4586,C 0.1342,E1 5.5585,E2 398.6425} C_DIS
LIN {X 86.2205,Y 107.6117,Z 180,A 52.24,B 5.4586,C 0.1371,E1 5.5625,E2 400.4564} C_DIS
LIN {X 89.6495,Y 104.7721,Z 180,A 50.4524,B 5.4585,C 0.1396,E1 5.5663,E2 402.2366} C_DIS
LIN {X 92.9893,Y 101.8196,Z 180,A 48.6261,B 5.4584,C 0.1428,E1 5.5701,E2 404.06} C_DIS
LIN {X 96.2342,Y 98.7583,Z 180,A 46.8053,B 5.4583,C 0.146,E1 5.5738,E2 405.8771} C_DIS
LIN {X 99.3791,Y 95.5931,Z 180,A 44.9929,B 5.4583,C 0.1492,E1 5.5773,E2 407.6847} C_DIS
LIN {X 102.3776,Y 92.3743,Z 180,A 43.1956,B 5.4581,C 0.1527,E1 5.5807,E2 409.4787} C_DIS
LIN {X 105.3492,Y 88.9707,Z 180,A 41.3609,B 5.4581,C 0.1561,E1 5.584,E2 411.3087} C_DIS
LIN {X 108.1657,Y 85.5244,Z 180,A 39.5185,B 5.4579,C 0.1601,E1 5.5872,E2 413.1508} C_DIS
LIN {X 110.8087,Y 82.0706,Z 180,A 37.771,B 5.4578,C 0.1634,E1 5.5902,E2 414.8915} C_DIS
LIN {X 113.4422,Y 78.3907,Z 180,A 35.942,B 5.4577,C 0.1671,E1 5.5931,E2 416.7147} C_DIS
LIN {X 115.8797,Y 74.7403,Z 180,A 34.1249,B 5.4576,C 0.1713,E1 5.5959,E2 418.5317} C_DIS
LIN {X 118.2225,Y 70.9766,Z 180,A 32.3284,B 5.4574,C 0.1751,E1 5.5985,E2 420.3233} C_DIS
LIN {X 120.4203,Y 67.1803,Z 180,A 30.5485,B 5.4574,C 0.179,E1 5.6009,E2 422.0986} C_DIS
LIN {X 122.3562,Y 63.5829,Z 180,A 28.9865,B 5.4572,C 0.1813,E1 5.6029,E2 423.6444} C_DIS
LIN {X 124.046,Y 60.2232,Z 180,A 27.4755,B 5.4572,C 0.1845,E1 5.6048,E2 425.1497} C_DIS
LIN {X 125.343,Y 57.4701,Z 180,A 26.2125,B 5.457,C 0.1878,E1 5.6063,E2 426.4131} C_DIS
LIN {X 126.9077,Y 53.932,Z 180,A 24.6741,B 5.457,C 0.1909,E1 5.608,E2 427.9438} C_DIS
LIN {X 128.2105,Y 50.7574,Z 180,A 23.2843,B 5.4568,C 0.1942,E1 5.6095,E2 429.3298} C_DIS
LIN {X 129.4277,Y 47.5678,Z 180,A 21.9016,B 5.4567,C 0.1974,E1 5.6108,E2 430.7087} C_DIS
LIN {X 130.3803,Y 44.8842,Z 180,A 20.758,B 5.4566,C 0.2,E1 5.6119,E2 431.848} C_DIS
LIN {X 131.4516,Y 41.6426,Z 180,A 19.3601,B 5.4565,C 0.2035,E1 5.6131,E2 433.2441} C_DIS
LIN {X 132.4588,Y 38.3195,Z 180,A 17.9653,B 5.4563,C 0.2067,E1 5.6142,E2 434.6337} C_DIS
LIN {X 133.3498,Y 35.0938,Z 180,A 16.5823,B 5.4562,C 0.2105,E1 5.6152,E2 436.0166} C_DIS
LIN {X 134.2439,Y 31.5091,Z 180,A 15.1131,B 5.4561,C 0.2137,E1 5.6161,E2 437.4785} C_DIS
LIN {X 134.9575,Y 28.2968,Z 180,A 13.7825,B 5.4559,C 0.217,E1 5.6169,E2 438.8054} C_DIS
LIN {X 135.5204,Y 25.4558,Z 180,A 12.587,B 5.4559,C 0.2202,E1 5.6175,E2 440.0006} C_DIS
LIN {X 136.1427,Y 21.8952,Z 180,A 11.1502,B 5.4557,C 0.2234,E1 5.6182,E2 441.4303} C_DIS
LIN {X 136.6167,Y 18.7113,Z 180,A 9.8492,B 5.4555,C 0.2267,E1 5.6187,E2 442.7276} C_DIS
LIN {X 137.0134,Y 15.5422,Z 180,A 8.5582,B 5.4555,C 0.2299,E1 5.6191,E2 444.0149} C_DIS
LIN {X 137.3343,Y 12.3902,Z 180,A 7.2778,B 5.4553,C 0.233,E1 5.6195,E2 445.2917} C_DIS
LIN {X 137.581,Y 9.2578,Z 180,A 6.0086,B 5.4551,C 0.2362,E1 5.6197,E2 446.5572} C_DIS
LIN {X 137.755,Y 6.1473,Z 180,A 4.7496,B 5.4551,C 0.2393,E1 5.6199,E2 447.8127} C_DIS
LIN {X 137.8837,Y 1.527,Z 180,A 2.9097,B 5.4548,C 0.2436,E1 5.62,E2 449.6437} C_DIS
LIN {X 137.8841,Y -1.468,Z 180,A 1.6775,B 5.4547,C 0.247,E1 5.62,E2 450.8754} C_DIS
LIN {X 137.755,Y -6.1473,Z 180,A -0.2294,B 5.4544,C 0.2519,E1 5.6199,E2 452.779} C_DIS
LIN {X 137.581,Y -9.2578,Z 180,A -1.493,B 5.4543,C 0.2551,E1 5.6196,E2 454.0396} C_DIS
LIN {X 137.3343,Y -12.3902,Z 180,A -2.7674,B 5.4541,C 0.2584,E1 5.6193,E2 455.3111} C_DIS
LIN {X 137.0134,Y -15.5422,Z 180,A -4.0523,B 5.454,C 0.2616,E1 5.619,E2 456.593} C_DIS
LIN {X 136.6167,Y -18.7113,Z 180,A -5.3475,B 5.4538,C 0.2649,E1 5.6185,E2 457.8852} C_DIS
LIN {X 136.1427,Y -21.8952,Z 180,A -6.6529,B 5.4537,C 0.2682,E1 5.6179,E2 459.1877} C_DIS
LIN {X 135.5901,Y -25.0913,Z 180,A -7.9686,B 5.4535,C 0.2715,E1 5.6173,E2 460.5003} C_DIS
LIN {X 135.0174,Y -28.0023,Z 180,A -9.1822,B 5.4533,C 0.2747,E1 5.6166,E2 461.7125} C_DIS
LIN {X 134.2562,Y -31.4552,Z 180,A -10.6066,B 5.4532,C 0.2781,E1 5.6157,E2 463.1325} C_DIS
LIN {X 133.4481,Y -34.7252,Z 180,A -11.9724,B 5.453,C 0.2815,E1 5.6148,E2 464.4952} C_DIS
LIN {X 132.5693,Y -37.9421,Z 180,A -13.325,B 5.4528,C 0.2848,E1 5.6138,E2 465.8447} C_DIS
LIN {X 131.6068,Y -41.157,Z 180,A -14.6866,B 5.4527,C 0.2881,E1 5.6127,E2 467.2034} C_DIS
LIN {X 130.5597,Y -44.3666,Z 180,A -16.0565,B 5.4525,C 0.2915,E1 5.6115,E2 468.5702} C_DIS
LIN {X 129.4277,Y -47.5678,Z 180,A -17.4343,B 5.4523,C 0.2948,E1 5.6102,E2 469.945} C_DIS
LIN {X 128.2105,Y -50.7574,Z 180,A -18.82,B 5.4521,C 0.2981,E1 5.6088,E2 471.3277} C_DIS
LIN {X 126.9077,Y -53.932,Z 180,A -20.213,B 5.4519,C 0.3014,E1 5.6073,E2 472.7178} C_DIS
LIN {X 125.5195,Y -57.0884,Z 180,A -21.6129,B 5.4518,C 0.3047,E1 5.6057,E2 474.1147} C_DIS
LIN {X 124.046,Y -60.2232,Z 180,A -23.0195,B 5.4516,C 0.3079,E1 5.604,E2 475.5184} C_DIS
LIN {X 122.4874,Y -63.3331,Z 180,A -24.4324,B 5.4514,C 0.3111,E1 5.6022,E2 476.9284} C_DIS
LIN {X 121.096,Y -65.953,Z 180,A -25.7174,B 5.4512,C 0.3151,E1 5.6005,E2 478.2213} C_DIS
LIN {X 118.9399,Y -69.7663,Z 180,A -27.4978,B 5.4509,C 0.3191,E1 5.598,E2 479.9982} C_DIS
LIN {X 116.6543,Y -73.5244,Z 180,A -29.286,B 5.4507,C 0.323,E1 5.5954,E2 481.783} C_DIS
LIN {X 114.1977,Y -77.2847,Z 180,A -31.0974,B 5.4505,C 0.3267,E1 5.5926,E2 483.589} C_DIS
LIN {X 111.5972,Y -80.9945,Z 180,A -32.9219,B 5.4503,C 0.3303,E1 5.5897,E2 485.4076} C_DIS
LIN {X 108.932,Y -84.5451,Z 180,A -34.7284,B 5.45,C 0.334,E1 5.5866,E2 487.2108} C_DIS
LIN {X 106.1481,Y -88.0149,Z 180,A -36.5394,B 5.4498,C 0.3376,E1 5.5834,E2 489.0186} C_DIS
LIN {X 103.3691,Y -91.2627,Z 180,A -38.3139,B 5.4496,C 0.3416,E1 5.5802,E2 490.7944} C_DIS
LIN {X 100.2396,Y -94.6893,Z 180,A -40.1604,B 5.4494,C 0.3445,E1 5.5767,E2 492.6321} C_DIS
LIN {X 97.2615,Y -97.7458,Z 180,A -41.9464,B 5.4491,C 0.3484,E1 5.5732,E2 494.4213} C_DIS
LIN {X 94.0387,Y -100.8502,Z 180,A -43.7685,B 5.4489,C 0.3517,E1 5.5695,E2 496.2402} C_DIS
LIN {X 90.5925,Y -103.9569,Z 180,A -45.6276,B 5.4488,C 0.3545,E1 5.5656,E2 498.092} C_DIS
LIN {X 87.3451,Y -106.7,Z 180,A -47.401,B 5.4485,C 0.3579,E1 5.5618,E2 499.8678} C_DIS
LIN {X 83.698,Y -109.5842,Z 180,A -49.2614,B 5.4484,C 0.3605,E1 5.5577,E2 501.7206} C_DIS
LIN {X 80.2752,Y -112.1158,Z 180,A -51.0346,B 5.4482,C 0.3636,E1 5.5537,E2 503.4958} C_DIS
LIN {X 76.6358,Y -114.6342,Z 180,A -52.8439,B 5.448,C 0.3663,E1 5.5495,E2 505.3028} C_DIS
LIN {X 72.7775,Y -117.1217,Z 180,A -54.6881,B 5.4478,C 0.3685,E1 5.5452,E2 507.1403} C_DIS
LIN {X 69.0079,Y -119.3816,Z 180,A -56.4869,B 5.4477,C 0.371,E1 5.5409,E2 508.937} C_DIS
LIN {X 65.4152,Y -121.3875,Z 180,A -58.223,B 5.4475,C 0.3739,E1 5.5366,E2 510.6779} C_DIS
LIN {X 61.7815,Y -123.2773,Z 180,A -59.8035,B 5.4475,C 0.3746,E1 5.5327,E2 512.2438} C_DIS
LIN {X 58.6587,Y -124.7934,Z 180,A -61.2269,B 5.4473,C 0.3762,E1 5.5291,E2 513.6659} C_DIS
LIN {X 56.0613,Y -125.9789,Z 180,A -62.4034,B 5.4473,C 0.3776,E1 5.5262,E2 514.8419} C_DIS
LIN {X 52.68,Y -127.4306,Z 180,A -63.931,B 5.4471,C 0.3794,E1 5.5222,E2 516.3705} C_DIS
LIN {X 49.1642,Y -128.8298,Z 180,A -65.4624,B 5.447,C 0.3807,E1 5.5182,E2 517.8977} C_DIS
LIN {X 45.9685,Y -130.0044,Z 180,A -66.8612,B 5.4469,C 0.382,E1 5.5146,E2 519.2955} C_DIS
LIN {X 42.9884,Y -131.0187,Z 180,A -68.1486,B 5.4469,C 0.3831,E1 5.5112,E2 520.581} C_DIS
LIN {X 39.55,Y -132.0986,Z 180,A -69.6378,B 5.4467,C 0.3844,E1 5.5072,E2 522.0702} C_DIS
LIN {X 36.3337,Y -133.0192,Z 180,A -71.0143,B 5.4467,C 0.3854,E1 5.5035,E2 523.4459} C_DIS
LIN {X 33.1168,Y -133.8563,Z 180,A -72.3833,B 5.4466,C 0.3864,E1 5.4998,E2 524.8141} C_DIS
LIN {X 30.2602,Y -134.5291,Z 180,A -73.597,B 5.4466,C 0.3872,E1 5.4965,E2 526.0278} C_DIS
LIN {X 26.693,Y -135.2838,Z 180,A -75.0951,B 5.4465,C 0.3881,E1 5.4924,E2 527.5248} C_DIS
LIN {X 23.4919,Y -135.8763,Z 180,A -76.438,B 5.4465,C 0.3888,E1 5.4887,E2 528.8672} C_DIS
LIN {X 19.3451,Y -136.5261,Z 180,A -78.1696,B 5.4464,C 0.3896,E1 5.4839,E2 530.5981} C_DIS
LIN {X 16.2233,Y -136.9322,Z 180,A -79.5002,B 5.4463,C 0.3905,E1 5.4802,E2 531.9323} C_DIS
LIN {X 12.3902,Y -137.3343,Z 180,A -81.0629,B 5.4463,C 0.3907,E1 5.4759,E2 533.4909} C_DIS
LIN {X 9.2578,Y -137.581,Z 180,A -82.3617,B 5.4463,C 0.391,E1 5.4723,E2 534.7896} C_DIS
LIN {X 6.1473,Y -137.755,Z 180,A -83.6509,B 5.4463,C 0.3913,E1 5.4687,E2 536.0787} C_DIS
LIN {X 2.4534,Y -137.8683,Z 180,A -85.2288,B 5.4462,C 0.3921,E1 5.4642,E2 537.6628} C_DIS
LIN {X 2.4534,Y -137.8683,Z 180,A -85.2288,B 5.4462,C 0.3921,E1 5.4642,E2 537.6628} C_DIS
Enddeposition()
LIN {X 0.9844,Y -138.7882,Z 180,A -85.1759,B 5.3793,C 0.386,E1 5.3973,E2 537.5746} C_DIS
Startdeposition()
$VEL.CP = VEL_PRINT
LIN {X 5.0991,Y -138.6993,Z 180,A -83.3821,B 5.3794,C 0.3844,E1 5.4024,E2 535.7675} C_DIS
LIN {X 9.19,Y -138.4895,Z 180,A -81.6211,B 5.3795,C 0.383,E1 5.4073,E2 533.9963} C_DIS
LIN {X 13.2079,Y -138.1626,Z 180,A -80.0673,B 5.3795,C 0.3838,E1 5.4116,E2 532.4562} C_DIS
LIN {X 17.2822,Y -137.7144,Z 180,A -77.7535,B 5.3801,C 0.3749,E1 5.4183,E2 530.0585} C_DIS
LIN {X 22.4765,Y -136.9609,Z 180,A -76.4304,B 5.3794,C 0.3848,E1 5.4216,E2 528.8467} C_DIS
LIN {X 25.0474,Y -136.5149,Z 180,A -75.2152,B 5.3796,C 0.3823,E1 5.425,E2 527.6125} C_DIS
LIN {X 28.2833,Y -135.8814,Z 180,A -73.8049,B 5.3796,C 0.3807,E1 5.4289,E2 526.1949} C_DIS
LIN {X 33.5309,Y -134.6825,Z 180,A -71.5771,B 5.3798,C 0.3789,E1 5.4349,E2 523.965} C_DIS
LIN {X 37.162,Y -133.7248,Z 180,A -69.9687,B 5.38,C 0.3768,E1 5.4393,E2 522.3478} C_DIS
LIN {X 40.8216,Y -132.6534,Z 180,A -68.5299,B 5.38,C 0.3771,E1 5.4431,E2 520.9259} C_DIS
LIN {X 44.1162,Y -131.5945,Z 180,A -67.1185,B 5.38,C 0.3759,E1 5.4468,E2 519.5158} C_DIS
LIN {X 47.358,Y -130.4629,Z 180,A -65.6735,B 5.3802,C 0.374,E1 5.4507,E2 518.0661} C_DIS
LIN {X 50.5209,Y -129.2709,Z 180,A -64.3347,B 5.3802,C 0.3732,E1 5.4541,E2 516.7339} C_DIS
LIN {X 53.7316,Y -127.9697,Z 180,A -62.9055,B 5.3803,C 0.3715,E1 5.4578,E2 515.3038} C_DIS
LIN {X 56.7546,Y -126.6577,Z 180,A -61.5806,B 5.3804,C 0.3703,E1 5.4612,E2 513.9826} C_DIS
LIN {X 60.0993,Y -125.1056,Z 180,A -60.054,B 5.3806,C 0.3682,E1 5.4651,E2 512.4543} C_DIS
LIN {X 63.3201,Y -123.5069,Z 180,A -58.5932,B 5.3806,C 0.3665,E1 5.4687,E2 510.9954} C_DIS
LIN {X 66.6318,Y -121.754,Z 180,A -56.8302,B 5.381,C 0.3612,E1 5.4731,E2 509.2026} C_DIS
LIN {X 71.6356,Y -118.8789,Z 180,A -54.7396,B 5.381,C 0.3617,E1 5.478,E2 507.1488} C_DIS
LIN {X 74.9997,Y -116.7856,Z 180,A -53.0453,B 5.3812,C 0.3582,E1 5.4821,E2 505.4454} C_DIS
LIN {X 78.7305,Y -114.3038,Z 180,A -50.8699,B 5.3818,C 0.3504,E1 5.4872,E2 503.2252} C_DIS
LIN {X 82.0459,Y -111.9477,Z 180,A -49.5076,B 5.3816,C 0.352,E1 5.4902,E2 501.9037} C_DIS
LIN {X 86.6689,Y -108.4084,Z 180,A -47.4412,B 5.3816,C 0.3524,E1 5.4947,E2 499.8799} C_DIS
LIN {X 88.941,Y -106.5524,Z 180,A -45.8058,B 5.3822,C 0.344,E1 5.4983,E2 498.1873} C_DIS
LIN {X 91.4275,Y -104.4263,Z 180,A -44.7171,B 5.3821,C 0.3452,E1 5.5005,E2 497.1321} C_DIS
LIN {X 94.5274,Y -101.6286,Z 180,A -42.9711,B 5.3823,C 0.3414,E1 5.5041,E2 495.3818} C_DIS
LIN {X 97.8158,Y -98.4676,Z 180,A -41.1296,B 5.3825,C 0.3381,E1 5.5078,E2 493.5441} C_DIS
LIN {X 102.2952,Y -93.8054,Z 180,A -38.5191,B 5.3828,C 0.3333,E1 5.5128,E2 490.939} C_DIS
LIN {X 105.8034,Y -89.83,Z 180,A -36.3029,B 5.3832,C 0.328,E1 5.5168,E2 488.7173} C_DIS
LIN {X 109.3558,Y -85.4705,Z 180,A -34.149,B 5.3833,C 0.3252,E1 5.5206,E2 486.5835} C_DIS
LIN {X 111.2364,Y -83.0078,Z 180,A -32.9985,B 5.3833,C 0.3241,E1 5.5225,E2 485.4488} C_DIS
LIN {X 113.3829,Y -80.0507,Z 180,A -31.3992,B 5.3837,C 0.3192,E1 5.5251,E2 483.8362} C_DIS
LIN {X 115.7014,Y -76.6625,Z 180,A -29.6782,B 5.3839,C 0.3147,E1 5.5278,E2 482.1102} C_DIS
LIN {X 118.6066,Y -72.0858,Z 180,A -27.4917,B 5.3842,C 0.31,E1 5.531,E2 479.9285} C_DIS
LIN {X 120.8881,Y -68.1904,Z 180,A -25.6847,B 5.3844,C 0.3062,E1 5.5335,E2 478.1273} C_DIS
LIN {X 123.0438,Y -64.215,Z 180,A -23.9316,B 5.3846,C 0.3031,E1 5.5358,E2 476.3874} C_DIS
LIN {X 124.6289,Y -61.0818,Z 180,A -22.539,B 5.3848,C 0.3002,E1 5.5375,E2 475.0009} C_DIS
LIN {X 126.0897,Y -58.0061,Z 180,A -21.1654,B 5.385,C 0.297,E1 5.5391,E2 473.6303} C_DIS
LIN {X 127.5732,Y -54.6675,Z 180,A -19.7256,B 5.3851,C 0.2941,E1 5.5407,E2 472.1981} C_DIS
LIN {X 128.8207,Y -51.658,Z 180,A -18.4,B 5.3853,C 0.2908,E1 5.5421,E2 470.8739} C_DIS
LIN {X 130.1971,Y -48.0872,Z 180,A -16.8857,B 5.3855,C 0.2875,E1 5.5436,E2 469.3668} C_DIS
LIN {X 131.25,Y -45.1313,Z 180,A -15.5765,B 5.3857,C 0.2838,E1 5.5448,E2 468.0546} C_DIS
LIN {X 132.32,Y -41.8906,Z 180,A -14.0074,B 5.386,C 0.2775,E1 5.5462,E2 466.4633} C_DIS
LIN {X 133.8436,Y -36.7371,Z 180,A -12.0903,B 5.386,C 0.276,E1 5.5476,E2 464.5838} C_DIS
LIN {X 134.5506,Y -34.0507,Z 180,A -10.9558,B 5.3862,C 0.273,E1 5.5484,E2 463.4498} C_DIS
LIN {X 135.37,Y -30.6323,Z 180,A -9.4632,B 5.3865,C 0.2683,E1 5.5494,E2 461.9506} C_DIS
LIN {X 136.2829,Y -26.2742,Z 180,A -7.6966,B 5.3867,C 0.2643,E1 5.5503,E2 460.1918} C_DIS
LIN {X 136.9799,Y -22.3627,Z 180,A -5.8343,B 5.387,C 0.2562,E1 5.5512,E2 458.2992} C_DIS
LIN {X 137.5094,Y -18.8449,Z 180,A -4.7293,B 5.387,C 0.2577,E1 5.5516,E2 457.2405} C_DIS
LIN {X 137.9568,Y -15.2118,Z 180,A -3.1834,B 5.3872,C 0.2528,E1 5.5521,E2 455.6887} C_DIS
LIN {X 138.3626,Y -10.9411,Z 180,A -1.3884,B 5.3874,C 0.2474,E1 5.5525,E2 453.8892} C_DIS
LIN {X 138.615,Y -7.0188,Z 180,A 0.1059,B 5.3876,C 0.2448,E1 5.5528,E2 452.4103} C_DIS
LIN {X 138.7636,Y -2.8981,Z 180,A 1.825,B 5.3878,C 0.2397,E1 5.5529,E2 450.6878} C_DIS
LIN {X 138.7859,Y 1.5593,Z 180,A 3.5845,B 5.388,C 0.2357,E1 5.5529,E2 448.9374} C_DIS
LIN {X 138.6892,Y 5.3574,Z 180,A 5.0546,B 5.3881,C 0.2327,E1 5.5528,E2 447.4788} C_DIS
LIN {X 138.5173,Y 8.7398,Z 180,A 6.4314,B 5.3883,C 0.229,E1 5.5525,E2 446.1036} C_DIS
LIN {X 138.1785,Y 13.043,Z 180,A 8.6867,B 5.3888,C 0.2167,E1 5.552,E2 443.7856} C_DIS
LIN {X 137.6469,Y 17.7974,Z 180,A 10.7053,B 5.389,C 0.2105,E1 5.5512,E2 441.7599} C_DIS
LIN {X 136.8646,Y 23.0533,Z 180,A 12.2437,B 5.3889,C 0.2144,E1 5.5506,E2 440.3052} C_DIS
LIN {X 135.6717,Y 29.2662,Z 180,A 14.7659,B 5.3891,C 0.2084,E1 5.5492,E2 437.7928} C_DIS
LIN {X 134.8461,Y 32.8626,Z 180,A 16.2077,B 5.3892,C 0.2054,E1 5.5483,E2 436.3605} C_DIS
LIN {X 134.044,Y 35.9938,Z 180,A 17.5406,B 5.3893,C 0.2018,E1 5.5473,E2 435.027} C_DIS
LIN {X 133.1138,Y 39.295,Z 180,A 18.9413,B 5.3895,C 0.1981,E1 5.5462,E2 433.6275} C_DIS
LIN {X 131.8495,Y 43.3505,Z 180,A 20.6935,B 5.3897,C 0.1934,E1 5.5447,E2 431.8744} C_DIS
LIN {X 130.617,Y 46.9307,Z 180,A 22.5439,B 5.39,C 0.1849,E1 5.543,E2 429.9861} C_DIS
LIN {X 129.223,Y 50.6442,Z 180,A 24.4503,B 5.3902,C 0.1765,E1 5.541,E2 428.044} C_DIS
LIN {X 127.0158,Y 55.9539,Z 180,A 26.0351,B 5.39,C 0.1822,E1 5.5393,E2 426.5597} C_DIS
LIN {X 125.138,Y 60.0314,Z 180,A 27.8999,B 5.3902,C 0.1772,E1 5.5371,E2 424.6925} C_DIS
LIN {X 123.3501,Y 63.6281,Z 180,A 29.5526,B 5.3903,C 0.1731,E1 5.535,E2 423.0398} C_DIS
LIN {X 121.2163,Y 67.6061,Z 180,A 32.2711,B 5.3909,C 0.1558,E1 5.5312,E2 420.2104} C_DIS
LIN {X 117.6074,Y 73.7051,Z 180,A 34.1703,B 5.3906,C 0.1638,E1 5.5286,E2 418.442} C_DIS
LIN {X 115.2867,Y 77.2841,Z 180,A 35.8228,B 5.3907,C 0.1612,E1 5.5261,E2 416.8026} C_DIS
LIN {X 113.1869,Y 80.3286,Z 180,A 37.5059,B 5.3909,C 0.1554,E1 5.5234,E2 415.0992} C_DIS
LIN {X 110.483,Y 84.0086,Z 180,A 39.366,B 5.3909,C 0.1514,E1 5.5203,E2 413.2416} C_DIS
LIN {X 107.3555,Y 87.9694,Z 180,A 41.1422,B 5.3909,C 0.1512,E1 5.5172,E2 411.5037} C_DIS
LIN {X 105.2178,Y 90.5152,Z 180,A 42.6968,B 5.3912,C 0.1456,E1 5.5144,E2 409.9256} C_DIS
LIN {X 102.2762,Y 93.8264,Z 180,A 44.4858,B 5.3912,C 0.1423,E1 5.511,E2 408.1412} C_DIS
LIN {X 99.3657,Y 96.9041,Z 180,A 46.2236,B 5.3913,C 0.1388,E1 5.5077,E2 406.4044} C_DIS
LIN {X 95.693,Y 100.5321,Z 180,A 48.3232,B 5.3914,C 0.135,E1 5.5035,E2 404.3083} C_DIS
LIN {X 93.3423,Y 102.7182,Z 180,A 49.5695,B 5.3914,C 0.1335,E1 5.5009,E2 403.0718} C_DIS
LIN {X 90.2556,Y 105.4414,Z 180,A 51.2799,B 5.3915,C 0.1302,E1 5.4973,E2 401.3597} C_DIS
LIN {X 86.9089,Y 108.2161,Z 180,A 53.0351,B 5.3916,C 0.1275,E1 5.4935,E2 399.6093} C_DIS
LIN {X 83.3877,Y 110.952,Z 180,A 54.8686,B 5.3916,C 0.1244,E1 5.4894,E2 397.7765} C_DIS
LIN {X 76.4986,Y 115.8094,Z 180,A 58.3014,B 5.3918,C 0.1193,E1 5.4816,E2 394.3496} C_DIS
LIN {X 72.5934,Y 118.2962,Z 180,A 59.9795,B 5.3918,C 0.1195,E1 5.4777,E2 392.7008} C_DIS
LIN {X 69.6695,Y 120.0416,Z 180,A 61.5403,B 5.3918,C 0.1154,E1 5.4739,E2 391.1205} C_DIS
LIN {X 65.8471,Y 122.1802,Z 180,A 63.3647,B 5.3919,C 0.1126,E1 5.4694,E2 389.2941} C_DIS
LIN {X 61.359,Y 124.4922,Z 180,A 65.9504,B 5.3921,C 0.1032,E1 5.4628,E2 386.645} C_DIS
LIN {X 56.5779,Y 126.7367,Z 180,A 67.1147,B 5.3919,C 0.114,E1 5.4602,E2 385.6089} C_DIS
LIN {X 53.1498,Y 128.2126,Z 180,A 68.9709,B 5.392,C 0.1081,E1 5.4553,E2 383.7135} C_DIS
LIN {X 50.0338,Y 129.4602,Z 180,A 70.367,B 5.392,C 0.1065,E1 5.4516,E2 382.3163} C_DIS
LIN {X 46.7656,Y 130.6765,Z 180,A 71.7663,B 5.392,C 0.1055,E1 5.448,E2 380.9222} C_DIS
LIN {X 43.1136,Y 131.9281,Z 180,A 73.3387,B 5.3921,C 0.1043,E1 5.4438,E2 379.3529} C_DIS
LIN {X 40.204,Y 132.8424,Z 180,A 74.5903,B 5.3921,C 0.1033,E1 5.4405,E2 378.1024} C_DIS
LIN {X 36.879,Y 133.804,Z 180,A 76.012,B 5.3921,C 0.1023,E1 5.4367,E2 376.6819} C_DIS
LIN {X 33.3566,Y 134.7267,Z 180,A 77.7746,B 5.3922,C 0.0979,E1 5.4318,E2 374.8872} C_DIS
LIN {X 24.6613,Y 136.584,Z 180,A 80.9383,B 5.3922,C 0.102,E1 5.4233,E2 371.788} C_DIS
LIN {X 15.9551,Y 137.8732,Z 180,A 84.6723,B 5.3922,C 0.0991,E1 5.413,E2 368.0431} C_DIS
LIN {X 13.2323,Y 138.1603,Z 180,A 85.8774,B 5.3922,C 0.0978,E1 5.4096,E2 366.829} C_DIS
LIN {X 10.017,Y 138.4306,Z 180,A 87.2508,B 5.3922,C 0.097,E1 5.4058,E2 365.4509} C_DIS
LIN {X 6.5014,Y 138.641,Z 180,A 88.7787,B 5.3922,C 0.0958,E1 5.4015,E2 363.9144} C_DIS
LIN {X 2.0995,Y 138.7769,Z 180,A 90.4975,B 5.3922,C 0.0968,E1 5.3967,E2 362.2087} C_DIS
LIN {X -1.0987,Y 138.7887,Z 180,A 91.9645,B 5.3922,C 0.095,E1 5.3926,E2 360.724} C_DIS
LIN {X -5.4602,Y 138.6852,Z 180,A 93.6651,B 5.3922,C 0.0963,E1 5.3879,E2 359.0367} C_DIS
LIN {X -11.7166,Y 138.2971,Z 180,A 96.5222,B 5.3923,C 0.0936,E1 5.3798,E2 356.1473} C_DIS
LIN {X -15.0185,Y 137.9776,Z 180,A 97.6352,B 5.3923,C 0.0969,E1 5.3768,E2 355.0671} C_DIS
LIN {X -18.5244,Y 137.5516,Z 180,A 99.3296,B 5.3923,C 0.0947,E1 5.372,E2 353.3439} C_DIS
LIN {X -23.242,Y 136.8331,Z 180,A 100.8934,B 5.3922,C 0.1001,E1 5.3679,E2 351.8319} C_DIS
LIN {X -25.7298,Y 136.387,Z 180,A 102.1498,B 5.3922,C 0.0982,E1 5.3643,E2 350.5496} C_DIS
LIN {X -29.4775,Y 135.6261,Z 180,A 103.7174,B 5.3922,C 0.0992,E1 5.3601,E2 348.9842} C_DIS
LIN {X -32.9222,Y 134.8318,Z 180,A 105.2633,B 5.3922,C 0.0992,E1 5.3558,E2 347.4285} C_DIS
LIN {X -37.7735,Y 133.5538,Z 180,A 107.1475,B 5.3922,C 0.1027,E1 5.3508,E2 345.5689} C_DIS
LIN {X -40.8582,Y 132.6422,Z 180,A 108.5894,B 5.3922,C 0.1025,E1 5.3469,E2 344.1136} C_DIS
LIN {X -44.3012,Y 131.5329,Z 180,A 110.0655,B 5.3922,C 0.1039,E1 5.343,E2 342.6406} C_DIS
LIN {X -47.3196,Y 130.4768,Z 180,A 111.4517,B 5.3922,C 0.1044,E1 5.3394,E2 341.247} C_DIS
LIN {X -55.6774,Y 127.1365,Z 180,A 115.2602,B 5.392,C 0.1074,E1 5.3295,E2 337.4297} C_DIS
LIN {X -61.1092,Y 124.6154,Z 180,A 117.4609,B 5.392,C 0.1131,E1 5.324,E2 335.2646} C_DIS
LIN {X -64.8323,Y 122.7197,Z 180,A 119.3931,B 5.392,C 0.1131,E1 5.3192,E2 333.3079} C_DIS
LIN {X -68.4534,Y 120.7397,Z 180,A 121.2504,B 5.392,C 0.1139,E1 5.3146,E2 331.4327} C_DIS
LIN {X -72.3845,Y 118.4244,Z 180,A 123.1602,B 5.3919,C 0.1164,E1 5.31,E2 329.5211} C_DIS
LIN {X -76.3936,Y 115.8785,Z 180,A 125.0955,B 5.3918,C 0.1196,E1 5.3055,E2 327.5904} C_DIS
LIN {X -79.9991,Y 113.4193,Z 180,A 127.0465,B 5.3918,C 0.121,E1 5.301,E2 325.6221} C_DIS
LIN {X -83.6656,Y 110.7424,Z 180,A 128.7953,B 5.3917,C 0.1254,E1 5.2971,E2 323.8906} C_DIS
LIN {X -86.8697,Y 108.2477,Z 180,A 130.6003,B 5.3917,C 0.127,E1 5.2931,E2 322.0708} C_DIS
LIN {X -90.4812,Y 105.2472,Z 180,A 132.6398,B 5.3916,C 0.1296,E1 5.2887,E2 320.0202} C_DIS
LIN {X -94.6513,Y 101.5132,Z 180,A 134.6738,B 5.3914,C 0.1367,E1 5.2846,E2 318.0228} C_DIS
LIN {X -97.1671,Y 99.1077,Z 180,A 136.3408,B 5.3914,C 0.1373,E1 5.2812,E2 316.3282} C_DIS
LIN {X -100.3631,Y 95.8699,Z 180,A 138.38,B 5.3914,C 0.1395,E1 5.2772,E2 314.2703} C_DIS
LIN {X -103.9867,Y 91.927,Z 180,A 140.4963,B 5.3912,C 0.1451,E1 5.2733,E2 312.1678} C_DIS
LIN {X -106.9026,Y 88.5191,Z 180,A 142.4017,B 5.3911,C 0.1486,E1 5.2698,E2 310.2572} C_DIS
LIN {X -109.7939,Y 84.9066,Z 180,A 144.4127,B 5.391,C 0.1519,E1 5.2663,E2 308.2351} C_DIS
LIN {X -112.5484,Y 81.2203,Z 180,A 146.281,B 5.3908,C 0.1566,E1 5.2633,E2 306.3725} C_DIS
LIN {X -115.1354,Y 77.5098,Z 180,A 148.2249,B 5.3908,C 0.1602,E1 5.2602,E2 304.4205} C_DIS
LIN {X -117.4982,Y 73.8785,Z 180,A 150.0166,B 5.3906,C 0.1645,E1 5.2575,E2 302.63} C_DIS
LIN {X -119.6063,Y 70.4142,Z 180,A 151.7655,B 5.3906,C 0.1679,E1 5.255,E2 300.8731} C_DIS
LIN {X -121.8548,Y 66.4471,Z 180,A 154.1352,B 5.3905,C 0.1681,E1 5.2517,E2 298.4433} C_DIS
LIN {X -123.9731,Y 62.4044,Z 180,A 155.5166,B 5.3902,C 0.1775,E1 5.25,E2 297.1273} C_DIS
LIN {X -125.5244,Y 59.2226,Z 180,A 157.0202,B 5.3901,C 0.1809,E1 5.2482,E2 295.6197} C_DIS
LIN {X -127.1537,Y 55.6378,Z 180,A 158.7667,B 5.39,C 0.184,E1 5.2462,E2 293.8592} C_DIS
LIN {X -129.8742,Y 48.9494,Z 180,A 161.5294,B 5.3896,C 0.1939,E1 5.2434,E2 291.1268} C_DIS
LIN {X -131.1789,Y 45.3363,Z 180,A 163.3781,B 5.3896,C 0.1958,E1 5.2416,E2 289.2463} C_DIS
LIN {X -132.2162,Y 42.2157,Z 180,A 164.7931,B 5.3895,C 0.1989,E1 5.2404,E2 287.8252} C_DIS
LIN {X -133.314,Y 38.6112,Z 180,A 166.3526,B 5.3893,C 0.2032,E1 5.2391,E2 286.2665} C_DIS
LIN {X -134.1572,Y 35.5693,Z 180,A 167.7229,B 5.3892,C 0.2061,E1 5.2381,E2 284.8887} C_DIS
LIN {X -134.9982,Y 32.2316,Z 180,A 169.1475,B 5.389,C 0.21,E1 5.2372,E2 283.4648} C_DIS
LIN {X -135.7928,Y 28.7051,Z 180,A 171.2012,B 5.389,C 0.2092,E1 5.236,E2 281.3408} C_DIS
LIN {X -136.6215,Y 24.4517,Z 180,A 172.5341,B 5.3887,C 0.2183,E1 5.2353,E2 280.0676} C_DIS
LIN {X -137.1594,Y 21.2284,Z 180,A 173.9263,B 5.3886,C 0.2217,E1 5.2347,E2 278.6711} C_DIS
LIN {X -137.6642,Y 17.6651,Z 180,A 175.4484,B 5.3884,C 0.2256,E1 5.2341,E2 277.1455} C_DIS
LIN {X -138.1845,Y 12.9805,Z 180,A 177.7919,B 5.3884,C 0.2276,E1 5.2335,E2 274.7527} C_DIS
LIN {X -138.4835,Y 9.2883,Z 180,A 179.1551,B 5.3881,C 0.2334,E1 5.2332,E2 273.412} C_DIS
LIN {X -138.7057,Y 4.9336,Z 180,A -179.1503,B 5.3878,C 0.2394,E1 5.233,E2 271.7323} C_DIS
LIN {X -138.7913,Y -0.7851,Z 180,A -176.5362,B 5.3876,C 0.2439,E1 5.233,E2 269.0876} C_DIS
LIN {X -138.6535,Y -6.253,Z 180,A -174.2743,B 5.3873,C 0.2503,E1 5.2332,E2 266.8269} C_DIS
LIN {X -138.4299,Y -10.0271,Z 180,A -172.757,B 5.3871,C 0.2551,E1 5.2334,E2 265.3163} C_DIS
LIN {X -138.0282,Y -14.5488,Z 180,A -170.9141,B 5.3868,C 0.2607,E1 5.2339,E2 263.4787} C_DIS
LIN {X -137.6088,Y -18.0879,Z 180,A -169.3202,B 5.3867,C 0.2637,E1 5.2345,E2 261.8701} C_DIS
LIN {X -137.1206,Y -21.4791,Z 180,A -167.9043,B 5.3865,C 0.2677,E1 5.2351,E2 260.455} C_DIS
LIN {X -136.5434,Y -24.8884,Z 180,A -166.4177,B 5.3863,C 0.2712,E1 5.2358,E2 258.9617} C_DIS
LIN {X -135.9436,Y -27.9779,Z 180,A -165.1188,B 5.3861,C 0.2748,E1 5.2365,E2 257.6638} C_DIS
LIN {X -135.2248,Y -31.268,Z 180,A -163.6032,B 5.386,C 0.2775,E1 5.2374,E2 256.1329} C_DIS
LIN {X -134.1619,Y -35.5519,Z 180,A -161.7172,B 5.3858,C 0.2819,E1 5.2388,E2 254.2398} C_DIS
LIN {X -133.0652,Y -39.4608,Z 180,A -160.0819,B 5.3855,C 0.2868,E1 5.24,E2 252.6107} C_DIS
LIN {X -132.0699,Y -42.6736,Z 180,A -158.5285,B 5.3854,C 0.289,E1 5.2414,E2 251.0368} C_DIS
LIN {X -130.1959,Y -48.0905,Z 180,A -156.3081,B 5.385,C 0.2967,E1 5.2434,E2 248.8367} C_DIS
LIN {X -129.2617,Y -50.5444,Z 180,A -155.0924,B 5.3849,C 0.2983,E1 5.2446,E2 247.6045} C_DIS
LIN {X -127.9237,Y -53.8416,Z 180,A -153.6135,B 5.3847,C 0.302,E1 5.2462,E2 246.125} C_DIS
LIN {X -126.3607,Y -57.4185,Z 180,A -151.952,B 5.3845,C 0.3057,E1 5.2481,E2 244.458} C_DIS
LIN {X -125.1343,Y -60.0392,Z 180,A -150.7075,B 5.3843,C 0.3083,E1 5.2496,E2 243.2074} C_DIS
LIN {X -123.2878,Y -63.7504,Z 180,A -148.5158,B 5.3843,C 0.308,E1 5.2525,E2 240.954} C_DIS
LIN {X -121.3305,Y -67.3998,Z 180,A -147.3467,B 5.3838,C 0.3174,E1 5.254,E2 239.8561} C_DIS
LIN {X -119.6891,Y -70.2733,Z 180,A -145.74,B 5.3838,C 0.3184,E1 5.2563,E2 238.2188} C_DIS
LIN {X -117.4316,Y -73.984,Z 180,A -143.8969,B 5.3835,C 0.3221,E1 5.259,E2 236.3699} C_DIS
LIN {X -115.1444,Y -77.4965,Z 180,A -142.099,B 5.3833,C 0.3255,E1 5.2618,E2 234.5638} C_DIS
LIN {X -112.5085,Y -81.2754,Z 180,A -139.9573,B 5.3832,C 0.3275,E1 5.2653,E2 232.3914} C_DIS
LIN {X -110.4564,Y -84.0429,Z 180,A -138.9041,B 5.3828,C 0.3342,E1 5.267,E2 231.387} C_DIS
LIN {X -108.219,Y -86.9053,Z 180,A -137.1948,B 5.3828,C 0.3354,E1 5.27,E2 229.6507} C_DIS
LIN {X -105.4507,Y -90.2448,Z 180,A -135.3383,B 5.3825,C 0.3386,E1 5.2734,E2 227.7862} C_DIS
LIN {X -102.4973,Y -93.5856,Z 180,A -133.4717,B 5.3823,C 0.3421,E1 5.2768,E2 225.9167} C_DIS
LIN {X -99.3563,Y -96.9137,Z 180,A -131.5368,B 5.3821,C 0.3454,E1 5.2806,E2 223.9762} C_DIS
LIN {X -96.1648,Y -100.0813,Z 180,A -129.6954,B 5.3818,C 0.3491,E1 5.2843,E2 222.1372} C_DIS
LIN {X -93.0421,Y -102.9905,Z 180,A -127.9119,B 5.3816,C 0.3521,E1 5.288,E2 220.3512} C_DIS
LIN {X -89.6949,Y -105.9183,Z 180,A -126.0212,B 5.3815,C 0.3548,E1 5.292,E2 218.4535} C_DIS
LIN {X -86.1937,Y -108.7866,Z 180,A -124.1137,B 5.3813,C 0.3575,E1 5.2961,E2 216.5411} C_DIS
LIN {X -78.545,Y -114.4311,Z 180,A -120.1693,B 5.3809,C 0.3636,E1 5.3051,E2 212.5945} C_DIS
LIN {X -74.3871,Y -117.1772,Z 180,A -118.3313,B 5.3805,C 0.3689,E1 5.3093,E2 210.7855} C_DIS
LIN {X -70.0966,Y -119.7928,Z 180,A -115.948,B 5.3805,C 0.3684,E1 5.3151,E2 208.3614} C_DIS
LIN {X -65.974,Y -122.112,Z 180,A -113.9868,B 5.3804,C 0.3708,E1 5.3199,E2 206.3991} C_DIS
LIN {X -58.8278,Y -125.7097,Z 180,A -110.4692,B 5.3803,C 0.3722,E1 5.3288,E2 202.8529} C_DIS
LIN {X -55.8871,Y -127.0457,Z 180,A -109.3803,B 5.38,C 0.3764,E1 5.3315,E2 201.7963} C_DIS
LIN {X -52.6,Y -128.4409,Z 180,A -107.8109,B 5.38,C 0.3767,E1 5.3356,E2 200.214} C_DIS
LIN {X -48.9047,Y -129.8909,Z 180,A -106.0554,B 5.38,C 0.3769,E1 5.3402,E2 198.4428} C_DIS
LIN {X -43.6889,Y -131.7368,Z 180,A -103.9207,B 5.3797,C 0.3804,E1 5.3458,E2 196.3274} C_DIS
LIN {X -39.8675,Y -132.9454,Z 180,A -102.2852,B 5.3797,C 0.3819,E1 5.3501,E2 194.6941} C_DIS
LIN {X -36.56,Y -133.8926,Z 180,A -100.809,B 5.3796,C 0.3821,E1 5.3541,E2 193.2101} C_DIS
LIN {X -27.9408,Y -135.9511,Z 180,A -97.3828,B 5.3793,C 0.3868,E1 5.3634,E2 189.8138} C_DIS
LIN {X -22.4554,Y -136.9644,Z 180,A -95.1541,B 5.3791,C 0.3886,E1 5.3695,E2 187.5943} C_DIS
LIN {X -19.9265,Y -137.3549,Z 180,A -93.7739,B 5.3794,C 0.385,E1 5.3734,E2 186.1709} C_DIS
LIN {X -16.4944,Y -137.8089,Z 180,A -92.3638,B 5.3794,C 0.3856,E1 5.3773,E2 184.7628} C_DIS
LIN {X -13.0468,Y -138.1781,Z 180,A -90.892,B 5.3794,C 0.3853,E1 5.3814,E2 183.285} C_DIS
LIN {X -8.8681,Y -138.5094,Z 180,A -89.1516,B 5.3794,C 0.3853,E1 5.3863,E2 181.5427} C_DIS
LIN {X -5.1812,Y -138.6961,Z 180,A -87.6945,B 5.3794,C 0.3861,E1 5.3903,E2 180.0937} C_DIS
LIN {X -1.2871,Y -138.7877,Z 180,A -85.9748,B 5.3794,C 0.3846,E1 5.3951,E2 178.3585} C_DIS
LIN {X -1.2871,Y -138.7877,Z 180,A -85.9748,B 5.3794,C 0.3846,E1 5.3951,E2 178.3585} C_DIS
Enddeposition()
LIN {X 0.988,Y -139.6903,Z 180,A -85.5346,B 5.3105,C 0.3926,E1 5.3279,E2 178.0358} C_DIS
Startdeposition()
$VEL.CP = VEL_PRINT
LIN {X -2.2407,Y -139.6774,Z 180,A -86.9727,B 5.3104,C 0.3942,E1 5.3238,E2 179.4897} C_DIS
LIN {X -5.4939,Y -139.5872,Z 180,A -88.3433,B 5.3104,C 0.3947,E1 5.32,E2 180.8656} C_DIS
LIN {X -9.4153,Y -139.3796,Z 180,A -90.0876,B 5.3102,C 0.3962,E1 5.315,E2 182.6283} C_DIS
LIN {X -13.3703,Y -139.0539,Z 180,A -91.5835,B 5.3104,C 0.3944,E1 5.3109,E2 184.1074} C_DIS
LIN {X -17.3009,Y -138.6217,Z 180,A -93.3088,B 5.3104,C 0.3953,E1 5.3061,E2 185.847} C_DIS
LIN {X -21.1326,Y -138.0876,Z 180,A -94.8463,B 5.3104,C 0.3943,E1 5.3019,E2 187.3785} C_DIS
LIN {X -24.2002,Y -137.5836,Z 180,A -96.2621,B 5.3103,C 0.3955,E1 5.2979,E2 188.8134} C_DIS
LIN {X -29.1445,Y -136.6214,Z 180,A -98.2055,B 5.3105,C 0.3932,E1 5.2926,E2 190.7413} C_DIS
LIN {X -34.2115,Y -135.4411,Z 180,A -100.725,B 5.3102,C 0.3964,E1 5.2857,E2 193.312} C_DIS
LIN {X -38.1592,Y -134.3832,Z 180,A -102.0444,B 5.3106,C 0.3913,E1 5.2822,E2 194.585} C_DIS
LIN {X -42.2651,Y -133.148,Z 180,A -103.7717,B 5.3107,C 0.3896,E1 5.2776,E2 196.3085} C_DIS
LIN {X -49.5131,Y -130.6269,Z 180,A -107.0449,B 5.3108,C 0.3884,E1 5.269,E2 199.5989} C_DIS
Enddeposition()
END
